   E6POS P1_B_1_App1Place={X 696.23437,Y 929.21517,Z 986.29988,A -180,B 0,C -180,S 2,T 2,E1 0,E2 0,E3 0,E4 0,E5 0,E6 0}
   E6POS P1_B_1_App2Place={X 696.23427,Y 929.21551,Z 786.30015,A -180,B 0,C 180,S 2,T 2,E1 0,E2 0,E3 0,E4 0,E5 0,E6 0}
   E6POS P1_B_1_Place={X 567.29912,Y 1052.67757,Z 666.29996,A -180,B 0,C 180,S 2,T 18,E1 0,E2 0,E3 0,E4 0,E5 0,E6 0}
   E6POS P1_B_2_App1Place={X 562.37046,Y 346.47969,Z 986.29988,A -180,B 0,C 180,S 2,T 2,E1 0,E2 0,E3 0,E4 0,E5 0,E6 0}
   E6POS P1_B_2_App2Place={X 562.37047,Y 346.47964,Z 786.30015,A -180,B 0,C 180,S 2,T 2,E1 0,E2 0,E3 0,E4 0,E5 0,E6 0}
   E6POS P1_B_2_Place={X 433.43516,Y 269.94251,Z 666.29996,A -180,B 0,C -180,S 2,T 2,E1 0,E2 0,E3 0,E4 0,E5 0,E6 0}
   E6POS P1_B_3_App1Place={X 4.05134,Y 173.92954,Z 986.29988,A 90,B 0,C 180,S 2,T 2,E1 0,E2 0,E3 0,E4 0,E5 0,E6 0}
   E6POS P1_B_3_App2Place={X 4.05139,Y 177.15339,Z 786.30015,A 90,B 0,C 180,S 2,T 2,E1 0,E2 0,E3 0,E4 0,E5 0,E6 0}
   E6POS P1_B_3_Place={X 134.71509,Y 273.89023,Z 666.29996,A 90,B 0,C 180,S 2,T 2,E1 0,E2 0,E3 0,E4 0,E5 0,E6 0}
   E6POS P1_B_4_App1Place={X 1006.46519,Y 1126.41051,Z 986.29988,A -90,B 0,C -180,S 2,T 2,E1 0,E2 0,E3 0,E4 0,E5 0,E6 0}
   E6POS P1_B_4_App2Place={X 1006.46535,Y 1126.41022,Z 786.30015,A -90,B 0,C 180,S 2,T 2,E1 0,E2 0,E3 0,E4 0,E5 0,E6 0}
   E6POS P1_B_4_Place={X 866.11759,Y 921.41578,Z 666.29996,A -90,B 0,C -180,S 2,T 2,E1 0,E2 0,E3 0,E4 0,E5 0,E6 0}
   E6POS P1_B_5_App1Place={X 696.22107,Y 346.20666,Z 986.29988,A -180,B 0,C -180,S 2,T 2,E1 0,E2 0,E3 0,E4 0,E5 0,E6 0}
   E6POS P1_B_5_App2Place={X 696.22108,Y 346.20663,Z 786.30015,A -180,B 0,C 180,S 2,T 2,E1 0,E2 0,E3 0,E4 0,E5 0,E6 0}
   E6POS P1_B_5_Place={X 567.29973,Y 269.67394,Z 666.29996,A -180,B 0,C 180,S 2,T 2,E1 0,E2 0,E3 0,E4 0,E5 0,E6 0}
   E6POS P1_B_6_App1Place={X 562.36978,Y 929.48243,Z 986.29988,A -180,B 0,C 180,S 2,T 2,E1 0,E2 0,E3 0,E4 0,E5 0,E6 0}
   E6POS P1_B_6_App2Place={X 562.36973,Y 929.48268,Z 786.30015,A -180,B 0,C -180,S 2,T 2,E1 0,E2 0,E3 0,E4 0,E5 0,E6 0}
   E6POS P1_B_6_Place={X 433.43554,Y 1052.93855,Z 666.29996,A -180,B 0,C 180,S 2,T 2,E1 0,E2 0,E3 0,E4 0,E5 0,E6 0}
   E6POS P1_B_7_App1Place={X 30.66561,Y 1051.60347,Z 986.29988,A -90,B 0,C 180,S 2,T 2,E1 0,E2 0,E3 0,E4 0,E5 0,E6 0}
   E6POS P1_B_7_App2Place={X 30.66561,Y 1051.60341,Z 786.30015,A -90,B 0,C 180,S 2,T 2,E1 0,E2 0,E3 0,E4 0,E5 0,E6 0}
   E6POS P1_B_7_Place={X 175.26087,Y 921.40676,Z 666.29996,A -90,B 0,C 180,S 2,T 2,E1 0,E2 0,E3 0,E4 0,E5 0,E6 0}
   E6POS P1_B_8_App1Place={X 955.95654,Y 159.58068,Z 986.29988,A 90,B 0,C 180,S 2,T 34,E1 0,E2 0,E3 0,E4 0,E5 0,E6 0}
   E6POS P1_B_8_App2Place={X 955.95654,Y 159.58069,Z 786.30015,A 90,B 0,C 180,S 2,T 34,E1 0,E2 0,E3 0,E4 0,E5 0,E6 0}
   E6POS P1_B_8_Place={X 825.57189,Y 273.90166,Z 666.29996,A 90,B 0,C 180,S 2,T 34,E1 0,E2 0,E3 0,E4 0,E5 0,E6 0}

   ;ENDFOLD
   ;FOLD  MosaicoC1_Pallet1

   E6POS P1_C1_1_App1Place={X 585.89482,Y 217.99128,Z 986.28312,A -180,B 0,C -180,S 2,T 2,E1 0,E2 0,E3 0,E4 0,E5 0,E6 0}
   E6POS P1_C1_1_App2Place={X 585.89477,Y 217.99161,Z 836.28257,A -180,B 0,C 180,S 2,T 2,E1 0,E2 0,E3 0,E4 0,E5 0,E6 0}
   E6POS P1_C1_1_Place={X 512.66253,Y 90.04064,Z 666.30129,A -180,B 0,C -180,S 2,T 2,E1 0,E2 0,E3 0,E4 0,E5 0,E6 0}
   E6POS P1_C1_2_App1Place={X 585.89508,Y 456.99119,Z 986.28312,A 180,B 0,C 180,S 2,T 2,E1 0,E2 0,E3 0,E4 0,E5 0,E6 0}
   E6POS P1_C1_2_App2Place={X 585.89505,Y 456.99134,Z 836.28257,A -180,B 0,C -180,S 2,T 2,E1 0,E2 0,E3 0,E4 0,E5 0,E6 0}
   E6POS P1_C1_2_Place={X 512.66375,Y 329.04071,Z 666.30129,A -180,B 0,C 180,S 2,T 2,E1 0,E2 0,E3 0,E4 0,E5 0,E6 0}
   E6POS P1_C1_3_App1Place={X 606.92676,Y 689.18267,Z 986.28312,A -180,B 0,C -180,S 2,T 2,E1 0,E2 0,E3 0,E4 0,E5 0,E6 0}
   E6POS P1_C1_3_App2Place={X 606.92684,Y 689.18232,Z 836.28257,A -180,B 0,C 180,S 2,T 2,E1 0,E2 0,E3 0,E4 0,E5 0,E6 0}
   E6POS P1_C1_3_Place={X 537.74298,Y 568.04115,Z 666.30129,A -180,B 0,C 180,S 2,T 2,E1 0,E2 0,E3 0,E4 0,E5 0,E6 0}
   E6POS P1_C1_4_App1Place={X 606.92634,Y 1021.18263,Z 986.28312,A 180,B 0,C -180,S 2,T 2,E1 0,E2 0,E3 0,E4 0,E5 0,E6 0}
   E6POS P1_C1_4_App2Place={X 606.92631,Y 1021.18275,Z 836.28257,A -180,B 0,C -180,S 2,T 2,E1 0,E2 0,E3 0,E4 0,E5 0,E6 0}
   E6POS P1_C1_4_Place={X 537.74306,Y 900.04115,Z 666.30129,A -180,B 0,C -180,S 2,T 18,E1 0,E2 0,E3 0,E4 0,E5 0,E6 0}
   E6POS P1_C1_5_App1Place={X 606.2009,Y 212.00378,Z 986.28312,A -180,B 0,C -180,S 2,T 2,E1 0,E2 0,E3 0,E4 0,E5 0,E6 0}
   E6POS P1_C1_5_App2Place={X 606.20094,Y 212.00353,Z 836.28257,A -180,B 0,C -180,S 2,T 2,E1 0,E2 0,E3 0,E4 0,E5 0,E6 0}
   E6POS P1_C1_5_Place={X 539.21738,Y 90.04103,Z 666.30129,A -180,B 0,C 180,S 2,T 2,E1 0,E2 0,E3 0,E4 0,E5 0,E6 0}
   E6POS P1_C1_6_App1Place={X 606.20038,Y 544.00374,Z 986.28312,A 180,B 0,C 180,S 2,T 2,E1 0,E2 0,E3 0,E4 0,E5 0,E6 0}
   E6POS P1_C1_6_App2Place={X 606.20036,Y 544.00384,Z 836.28257,A -180,B 0,C 180,S 2,T 2,E1 0,E2 0,E3 0,E4 0,E5 0,E6 0}
   E6POS P1_C1_6_Place={X 539.2172,Y 422.04157,Z 666.30129,A -180,B 0,C 180,S 2,T 2,E1 0,E2 0,E3 0,E4 0,E5 0,E6 0}
   E6POS P1_C1_7_App1Place={X 516.90957,Y 854.03849,Z 986.28312,A 180,B 0,C -180,S 2,T 2,E1 0,E2 0,E3 0,E4 0,E5 0,E6 0}
   E6POS P1_C1_7_App2Place={X 516.9096,Y 854.03829,Z 836.28257,A -180,B 0,C 180,S 2,T 2,E1 0,E2 0,E3 0,E4 0,E5 0,E6 0}
   E6POS P1_C1_7_Place={X 516.90992,Y 754.0383,Z 666.30129,A -180,B 0,C -180,S 2,T 2,E1 0,E2 0,E3 0,E4 0,E5 0,E6 0}
   E6POS P1_C1_8_App1Place={X 516.90957,Y 1093.03906,Z 986.28312,A -180,B 0,C -180,S 2,T 2,E1 0,E2 0,E3 0,E4 0,E5 0,E6 0}
   E6POS P1_C1_8_App2Place={X 516.90967,Y 1093.03859,Z 836.28257,A -180,B 0,C 180,S 2,T 2,E1 0,E2 0,E3 0,E4 0,E5 0,E6 0}
   E6POS P1_C1_8_Place={X 516.90982,Y 993.03884,Z 666.30129,A -180,B 0,C -180,S 2,T 2,E1 0,E2 0,E3 0,E4 0,E5 0,E6 0}

   ;ENDFOLD
   ;FOLD  MosaicoE1_Pallet1

   E6POS P1_E1_1_App1Place={X 194.85126,Y 240.03141,Z 993.17126,A 90,B 0,C 180,S 2,T 2,E1 0,E2 0,E3 0,E4 0,E5 0,E6 0}
   E6POS P1_E1_1_App2Place={X 194.85179,Y 240.03149,Z 843.1711,A 90,B 0,C 180,S 2,T 2,E1 0,E2 0,E3 0,E4 0,E5 0,E6 0}
   E6POS P1_E1_1_Place={X 73.35816,Y 240.03167,Z 690.47496,A 90,B 0,C 180,S 2,T 2,E1 0,E2 0,E3 0,E4 0,E5 0,E6 0}
   E6POS P1_E1_2_App1Place={X 522.85183,Y 240.03135,Z 993.17126,A 90,B 0,C 180,S 2,T 34,E1 0,E2 0,E3 0,E4 0,E5 0,E6 0}
   E6POS P1_E1_2_App2Place={X 522.85174,Y 240.03121,Z 843.1711,A 90,B 0,C 180,S 2,T 34,E1 0,E2 0,E3 0,E4 0,E5 0,E6 0}
   E6POS P1_E1_2_Place={X 401.35813,Y 240.03144,Z 690.47496,A 90,B 0,C 180,S 2,T 34,E1 0,E2 0,E3 0,E4 0,E5 0,E6 0}
   E6POS P1_E1_3_App1Place={X 850.85178,Y 240.03166,Z 993.17126,A 90,B 0,C 180,S 2,T 34,E1 0,E2 0,E3 0,E4 0,E5 0,E6 0}
   E6POS P1_E1_3_App2Place={X 850.85169,Y 240.03128,Z 843.1711,A 90,B 0,C 180,S 2,T 34,E1 0,E2 0,E3 0,E4 0,E5 0,E6 0}
   E6POS P1_E1_3_Place={X 729.35887,Y 240.0316,Z 690.47496,A 90,B 0,C 180,S 2,T 34,E1 0,E2 0,E3 0,E4 0,E5 0,E6 0}
   E6POS P1_E1_4_App1Place={X 622.32094,Y 1010.79553,Z 993.17126,A -180,B 0,C -180,S 2,T 2,E1 0,E2 0,E3 0,E4 0,E5 0,E6 0}
   E6POS P1_E1_4_App2Place={X 622.32108,Y 1010.79584,Z 843.1711,A -180,B 0,C 180,S 2,T 18,E1 0,E2 0,E3 0,E4 0,E5 0,E6 0}
   E6POS P1_E1_4_Place={X 622.32108,Y 907.44031,Z 690.47496,A -180,B 0,C 180,S 2,T 2,E1 0,E2 0,E3 0,E4 0,E5 0,E6 0}
   E6POS P1_E1_5_App1Place={X 622.32111,Y 907.44046,Z 993.17126,A -180,B 0,C 180,S 2,T 2,E1 0,E2 0,E3 0,E4 0,E5 0,E6 0}
   E6POS P1_E1_5_App2Place={X 676.32064,Y 907.52752,Z 843.1711,A -180,B 0,C 180,S 2,T 2,E1 0,E2 0,E3 0,E4 0,E5 0,E6 0}
   E6POS P1_E1_5_Place={X 676.32052,Y 907.52694,Z 690.47496,A -180,B 0,C 180,S 2,T 2,E1 0,E2 0,E3 0,E4 0,E5 0,E6 0}
   E6POS P1_E1_6_App1Place={X 676.32064,Y 907.52752,Z 993.17126,A -180,B 0,C 180,S 2,T 2,E1 0,E2 0,E3 0,E4 0,E5 0,E6 0}
   E6POS P1_E1_6_App2Place={X 730.3205,Y 907.52691,Z 843.1711,A -180,B 0,C 180,S 2,T 2,E1 0,E2 0,E3 0,E4 0,E5 0,E6 0}
   E6POS P1_E1_6_Place={X 730.32055,Y 907.52712,Z 690.47496,A -180,B 0,C 180,S 2,T 2,E1 0,E2 0,E3 0,E4 0,E5 0,E6 0}
   E6POS P1_E1_7_App1Place={X 730.3205,Y 907.52691,Z 993.17126,A -180,B 0,C 180,S 2,T 2,E1 0,E2 0,E3 0,E4 0,E5 0,E6 0}
   E6POS P1_E1_7_App2Place={X 784.32058,Y 907.52713,Z 843.1711,A -180,B 0,C 180,S 2,T 2,E1 0,E2 0,E3 0,E4 0,E5 0,E6 0}
   E6POS P1_E1_7_Place={X 784.32065,Y 907.52737,Z 690.47496,A -180,B 0,C 180,S 2,T 2,E1 0,E2 0,E3 0,E4 0,E5 0,E6 0}
   E6POS P1_E1_8_App1Place={X 624.31165,Y 190.79546,Z 993.17126,A -180,B 0,C 180,S 2,T 2,E1 0,E2 0,E3 0,E4 0,E5 0,E6 0}
   E6POS P1_E1_8_App2Place={X 624.31125,Y 190.79541,Z 843.1711,A -180,B 0,C 180,S 2,T 2,E1 0,E2 0,E3 0,E4 0,E5 0,E6 0}

   E6POS P1_E1_8_Place={X 624.31203,Y 87.43905,Z 690.47496,A -180,B 0,C 180,S 2,T 2,E1 0,E2 0,E3 0,E4 0,E5 0,E6 0}
   E6POS P1_E1_9_App1Place={X 624.31193,Y 87.4387,Z 993.17126,A -180,B 0,C 180,S 2,T 2,E1 0,E2 0,E3 0,E4 0,E5 0,E6 0}
   E6POS P1_E1_9_App2Place={X 678.31177,Y 87.43866,Z 843.1711,A -180,B 0,C 180,S 2,T 2,E1 0,E2 0,E3 0,E4 0,E5 0,E6 0}

   E6POS P1_E1_9_Place={X 678.31185,Y 87.43891,Z 690.47496,A -180,B 0,C -180,S 2,T 2,E1 0,E2 0,E3 0,E4 0,E5 0,E6 0}
   E6POS P1_E1_10_App1Place={X 678.31177,Y 87.43866,Z 993.17126,A -180,B 0,C 180,S 2,T 2,E1 0,E2 0,E3 0,E4 0,E5 0,E6 0}
   E6POS P1_E1_10_App2Place={X 732.31118,Y 87.43893,Z 843.1711,A -180,B 0,C 180,S 2,T 2,E1 0,E2 0,E3 0,E4 0,E5 0,E6 0}

   E6POS P1_E1_10_Place={X 732.31137,Y 87.43945,Z 690.47496,A -180,B 0,C 180,S 2,T 2,E1 0,E2 0,E3 0,E4 0,E5 0,E6 0}
   E6POS P1_E1_11_App1Place={X 732.31118,Y 87.43893,Z 993.17126,A -180,B 0,C 180,S 2,T 2,E1 0,E2 0,E3 0,E4 0,E5 0,E6 0}
   E6POS P1_E1_11_App2Place={X 786.31144,Y 87.43887,Z 843.1711,A -180,B 0,C -180,S 2,T 2,E1 0,E2 0,E3 0,E4 0,E5 0,E6 0}

   E6POS P1_E1_11_Place={X 786.31151,Y 87.43905,Z 690.47496,A -180,B 0,C -180,S 2,T 2,E1 0,E2 0,E3 0,E4 0,E5 0,E6 0}
   E6POS P1_E1_12_App1Place={X 838.55884,Y 1064.39297,Z 993.17126,A -90,B 0,C -180,S 2,T 2,E1 0,E2 0,E3 0,E4 0,E5 0,E6 0}
   E6POS P1_E1_12_App2Place={X 838.55901,Y 1064.39353,Z 843.1711,A -90,B 0,C 180,S 2,T 2,E1 0,E2 0,E3 0,E4 0,E5 0,E6 0}

   E6POS P1_E1_12_Place={X 938.55894,Y 964.39354,Z 690.47496,A -90,B 0,C 180,S 2,T 2,E1 0,E2 0,E3 0,E4 0,E5 0,E6 0}
   E6POS P1_E1_13_App1Place={X 510.55787,Y 1064.39363,Z 993.17126,A -89.99997,B 0,C 180,S 2,T 2,E1 0,E2 0,E3 0,E4 0,E5 0,E6 0}
   E6POS P1_E1_13_App2Place={X 510.55802,Y 1064.39347,Z 843.1711,A -89.99997,B 0,C 180,S 2,T 2,E1 0,E2 0,E3 0,E4 0,E5 0,E6 0}

   E6POS P1_E1_13_Place={X 610.5583,Y 964.39342,Z 690.47496,A -89.99997,B 0,C 180,S 2,T 2,E1 0,E2 0,E3 0,E4 0,E5 0,E6 0}
   E6POS P1_E1_14_App1Place={X 182.55908,Y 1064.39364,Z 993.17126,A -90,B 0,C 180,S 2,T 2,E1 0,E2 0,E3 0,E4 0,E5 0,E6 0}
   E6POS P1_E1_14_App2Place={X 182.55871,Y 1064.39336,Z 843.1711,A -90,B 0,C 180,S 2,T 2,E1 0,E2 0,E3 0,E4 0,E5 0,E6 0}

   E6POS P1_E1_14_Place={X 282.55806,Y 964.39307,Z 690.47496,A -89.99997,B 0,C 180,S 2,T 2,E1 0,E2 0,E3 0,E4 0,E5 0,E6 0}

   ;ENDFOLD
   ;FOLD  MosaicoE2_Pallet1

   E6POS P1_E2_1_App1Place={X 194.85126,Y 240.03141,Z 953.17126,A 90,B 0,C 180,S 2,T 2,E1 0,E2 0,E3 0,E4 0,E5 0,E6 0}
   E6POS P1_E2_1_App2Place={X 194.85179,Y 240.03149,Z 803.1711,A 90,B 0,C 180,S 2,T 2,E1 0,E2 0,E3 0,E4 0,E5 0,E6 0}
   E6POS P1_E2_1_Place={X 73.35816,Y 240.03167,Z 650.47496,A 90,B 0,C 180,S 2,T 2,E1 0,E2 0,E3 0,E4 0,E5 0,E6 0}
   E6POS P1_E2_2_App1Place={X 522.85183,Y 240.03135,Z 953.17126,A 90,B 0,C 180,S 2,T 34,E1 0,E2 0,E3 0,E4 0,E5 0,E6 0}
   E6POS P1_E2_2_App2Place={X 522.85174,Y 240.03121,Z 803.1711,A 90,B 0,C 180,S 2,T 34,E1 0,E2 0,E3 0,E4 0,E5 0,E6 0}
   E6POS P1_E2_2_Place={X 401.35813,Y 240.03144,Z 650.47496,A 90,B 0,C 180,S 2,T 34,E1 0,E2 0,E3 0,E4 0,E5 0,E6 0}
   E6POS P1_E2_3_App1Place={X 850.85178,Y 240.03166,Z 953.17126,A 90,B 0,C 180,S 2,T 34,E1 0,E2 0,E3 0,E4 0,E5 0,E6 0}
   E6POS P1_E2_3_App2Place={X 850.85169,Y 240.03128,Z 803.1711,A 90,B 0,C 180,S 2,T 34,E1 0,E2 0,E3 0,E4 0,E5 0,E6 0}
   E6POS P1_E2_3_Place={X 729.35887,Y 240.0316,Z 650.47496,A 90,B 0,C 180,S 2,T 34,E1 0,E2 0,E3 0,E4 0,E5 0,E6 0}
   E6POS P1_E2_4_App1Place={X 622.32094,Y 1010.79553,Z 953.17126,A -180,B 0,C -180,S 2,T 2,E1 0,E2 0,E3 0,E4 0,E5 0,E6 0}
   E6POS P1_E2_4_App2Place={X 622.32108,Y 1010.79584,Z 803.1711,A -180,B 0,C 180,S 2,T 18,E1 0,E2 0,E3 0,E4 0,E5 0,E6 0}
   E6POS P1_E2_4_Place={X 622.32108,Y 907.44031,Z 650.47496,A -180,B 0,C 180,S 2,T 18,E1 0,E2 0,E3 0,E4 0,E5 0,E6 0}
   E6POS P1_E2_5_App1Place={X 622.32111,Y 907.44046,Z 953.17126,A -180,B 0,C 180,S 2,T 2,E1 0,E2 0,E3 0,E4 0,E5 0,E6 0}
   E6POS P1_E2_5_App2Place={X 676.32064,Y 907.52752,Z 803.1711,A -180,B 0,C 180,S 2,T 2,E1 0,E2 0,E3 0,E4 0,E5 0,E6 0}
   E6POS P1_E2_5_Place={X 676.32052,Y 907.52694,Z 650.47496,A -180,B 0,C 180,S 2,T 18,E1 0,E2 0,E3 0,E4 0,E5 0,E6 0}
   E6POS P1_E2_6_App1Place={X 676.32064,Y 907.52752,Z 953.17126,A -180,B 0,C 180,S 2,T 2,E1 0,E2 0,E3 0,E4 0,E5 0,E6 0}
   E6POS P1_E2_6_App2Place={X 730.3205,Y 907.52691,Z 803.1711,A -180,B 0,C 180,S 2,T 2,E1 0,E2 0,E3 0,E4 0,E5 0,E6 0}
   E6POS P1_E2_6_Place={X 730.32055,Y 907.52712,Z 650.47496,A -180,B 0,C 180,S 2,T 2,E1 0,E2 0,E3 0,E4 0,E5 0,E6 0}
   E6POS P1_E2_7_App1Place={X 730.3205,Y 907.52691,Z 953.17126,A -180,B 0,C 180,S 2,T 2,E1 0,E2 0,E3 0,E4 0,E5 0,E6 0}
   E6POS P1_E2_7_App2Place={X 784.32058,Y 907.52713,Z 803.1711,A -180,B 0,C 180,S 2,T 2,E1 0,E2 0,E3 0,E4 0,E5 0,E6 0}
   E6POS P1_E2_7_Place={X 784.32065,Y 907.52737,Z 650.47496,A -180,B 0,C 180,S 2,T 2,E1 0,E2 0,E3 0,E4 0,E5 0,E6 0}
   E6POS P1_E2_8_App1Place={X 624.31165,Y 190.79546,Z 953.17126,A -180,B 0,C 180,S 2,T 2,E1 0,E2 0,E3 0,E4 0,E5 0,E6 0}
   E6POS P1_E2_8_App2Place={X 624.31125,Y 190.79541,Z 803.1711,A -180,B 0,C 180,S 2,T 2,E1 0,E2 0,E3 0,E4 0,E5 0,E6 0}
   E6POS P1_E2_8_Place={X 624.31203,Y 87.43905,Z 650.47496,A -180,B 0,C 180,S 2,T 2,E1 0,E2 0,E3 0,E4 0,E5 0,E6 0}
   E6POS P1_E2_9_App1Place={X 624.31193,Y 87.4387,Z 953.17126,A -180,B 0,C 180,S 2,T 2,E1 0,E2 0,E3 0,E4 0,E5 0,E6 0}
   E6POS P1_E2_9_App2Place={X 678.31177,Y 87.43866,Z 803.1711,A -180,B 0,C 180,S 2,T 2,E1 0,E2 0,E3 0,E4 0,E5 0,E6 0}
   E6POS P1_E2_9_Place={X 678.31185,Y 87.43891,Z 650.47496,A -180,B 0,C -180,S 2,T 2,E1 0,E2 0,E3 0,E4 0,E5 0,E6 0}
   E6POS P1_E2_10_App1Place={X 678.31177,Y 87.43866,Z 953.17126,A -180,B 0,C 180,S 2,T 2,E1 0,E2 0,E3 0,E4 0,E5 0,E6 0}
   E6POS P1_E2_10_App2Place={X 732.31118,Y 87.43893,Z 803.1711,A -180,B 0,C 180,S 2,T 2,E1 0,E2 0,E3 0,E4 0,E5 0,E6 0}
   E6POS P1_E2_10_Place={X 732.31137,Y 87.43945,Z 650.47496,A -180,B 0,C 180,S 2,T 2,E1 0,E2 0,E3 0,E4 0,E5 0,E6 0}
   E6POS P1_E2_11_App1Place={X 732.31118,Y 87.43893,Z 953.17126,A -180,B 0,C 180,S 2,T 2,E1 0,E2 0,E3 0,E4 0,E5 0,E6 0}
   E6POS P1_E2_11_App2Place={X 786.31144,Y 87.43887,Z 803.1711,A -180,B 0,C -180,S 2,T 2,E1 0,E2 0,E3 0,E4 0,E5 0,E6 0}
   E6POS P1_E2_11_Place={X 786.31151,Y 87.43905,Z 650.47496,A -180,B 0,C -180,S 2,T 2,E1 0,E2 0,E3 0,E4 0,E5 0,E6 0}
   E6POS P1_E2_12_App1Place={X 838.55884,Y 1064.39297,Z 953.17126,A -90,B 0,C -180,S 2,T 2,E1 0,E2 0,E3 0,E4 0,E5 0,E6 0}
   E6POS P1_E2_12_App2Place={X 838.55901,Y 1064.39353,Z 803.1711,A -90,B 0,C 180,S 2,T 2,E1 0,E2 0,E3 0,E4 0,E5 0,E6 0}

   E6POS P1_E2_12_Place={X 938.55894,Y 964.39354,Z 650.47496,A -90,B 0,C 180,S 2,T 2,E1 0,E2 0,E3 0,E4 0,E5 0,E6 0}
   E6POS P1_E2_13_App1Place={X 510.55787,Y 1064.39363,Z 953.17126,A -89.99997,B 0,C 180,S 2,T 2,E1 0,E2 0,E3 0,E4 0,E5 0,E6 0}
   E6POS P1_E2_13_App2Place={X 510.55802,Y 1064.39347,Z 803.1711,A -89.99997,B 0,C 180,S 2,T 2,E1 0,E2 0,E3 0,E4 0,E5 0,E6 0}

   E6POS P1_E2_13_Place={X 610.5583,Y 964.39342,Z 650.47496,A -89.99997,B 0,C 180,S 2,T 2,E1 0,E2 0,E3 0,E4 0,E5 0,E6 0}
   E6POS P1_E2_14_App1Place={X 182.55908,Y 1064.39364,Z 953.17126,A -90,B 0,C 180,S 2,T 2,E1 0,E2 0,E3 0,E4 0,E5 0,E6 0}
   E6POS P1_E2_14_App2Place={X 182.55871,Y 1064.39336,Z 803.1711,A -90,B 0,C 180,S 2,T 2,E1 0,E2 0,E3 0,E4 0,E5 0,E6 0}

   E6POS P1_E2_14_Place={X 282.55806,Y 964.39307,Z 650.47496,A -89.99997,B 0,C 180,S 2,T 2,E1 0,E2 0,E3 0,E4 0,E5 0,E6 0}

   ;ENDFOLD
   ;FOLD  MosaicoF_Pallet1

   E6POS P1_F_1_App1Place={X 185.70996,Y 503.84704,Z 990.17104,A -89.99997,B 0,C 180,S 2,T 2,E1 0,E2 0,E3 0,E4 0,E5 0,E6 0}
   E6POS P1_F_1_App2Place={X 185.71037,Y 503.84729,Z 840.17131,A -89.99997,B 0,C 180,S 2,T 2,E1 0,E2 0,E3 0,E4 0,E5 0,E6 0}
   E6POS P1_F_1_Place={X 59.05642,Y 604.23198,Z 654.93708,A -89.99997,B 0,C 180,S 2,T 2,E1 0,E2 0,E3 0,E4 0,E5 0,E6 0}
   E6POS P1_F_2_App1Place={X 484.71014,Y 503.84728,Z 990.17104,A -89.99997,B 0,C 180,S 2,T 2,E1 0,E2 0,E3 0,E4 0,E5 0,E6 0}
   E6POS P1_F_2_App2Place={X 484.71027,Y 503.84725,Z 840.17131,A -89.99997,B 0,C 180,S 2,T 2,E1 0,E2 0,E3 0,E4 0,E5 0,E6 0}
   E6POS P1_F_2_Place={X 358.05527,Y 604.23504,Z 654.93708,A -89.99997,B 0,C 180,S 2,T 2,E1 0,E2 0,E3 0,E4 0,E5 0,E6 0}
   E6POS P1_F_3_App1Place={X 783.33985,Y 500.30966,Z 990.17104,A -90,B 0,C 180,S 2,T 2,E1 0,E2 0,E3 0,E4 0,E5 0,E6 0}
   E6POS P1_F_3_App2Place={X 783.33995,Y 500.31005,Z 840.17131,A -90,B 0,C 180,S 2,T 2,E1 0,E2 0,E3 0,E4 0,E5 0,E6 0}
   E6POS P1_F_3_Place={X 657.05567,Y 600.73453,Z 654.93708,A -90,B 0,C 180,S 2,T 2,E1 0,E2 0,E3 0,E4 0,E5 0,E6 0}
   E6POS P1_F_4_App1Place={X 981.33967,Y 500.30989,Z 990.17104,A -90,B 0,C 180,S 2,T 2,E1 0,E2 0,E3 0,E4 0,E5 0,E6 0}
   E6POS P1_F_4_App2Place={X 981.33982,Y 500.30975,Z 840.17131,A -90,B 0,C 180,S 2,T 2,E1 0,E2 0,E3 0,E4 0,E5 0,E6 0}
   E6POS P1_F_4_Place={X 855.0547,Y 600.73492,Z 654.93708,A -90,B 0,C 180,S 2,T 2,E1 0,E2 0,E3 0,E4 0,E5 0,E6 0}
   E6POS P1_F_5_App1Place={X 185.3398,Y 495.81009,Z 990.17104,A -90,B 0,C 180,S 2,T 2,E1 0,E2 0,E3 0,E4 0,E5 0,E6 0}
   E6POS P1_F_5_App2Place={X 185.33937,Y 495.81034,Z 840.17131,A -90,B 0,C 180,S 2,T 2,E1 0,E2 0,E3 0,E4 0,E5 0,E6 0}
   E6POS P1_F_5_Place={X 59.05866,Y 596.22286,Z 654.93708,A -90,B 0,C 180,S 2,T 2,E1 0,E2 0,E3 0,E4 0,E5 0,E6 0}
   E6POS P1_F_6_App1Place={X 383.34027,Y 495.81061,Z 990.17104,A -90,B 0,C 180,S 2,T 2,E1 0,E2 0,E3 0,E4 0,E5 0,E6 0}
   E6POS P1_F_6_App2Place={X 383.33973,Y 495.81031,Z 840.17131,A -90,B 0,C 180,S 2,T 2,E1 0,E2 0,E3 0,E4 0,E5 0,E6 0}
   E6POS P1_F_6_Place={X 257.05855,Y 596.22277,Z 654.93708,A -90,B 0,C 180,S 2,T 2,E1 0,E2 0,E3 0,E4 0,E5 0,E6 0}
   E6POS P1_F_7_App1Place={X 581.71086,Y 500.34692,Z 990.17104,A -90,B 0,C 180,S 2,T 2,E1 0,E2 0,E3 0,E4 0,E5 0,E6 0}
   E6POS P1_F_7_App2Place={X 581.71089,Y 500.3468,Z 840.17131,A -90,B 0,C 180,S 2,T 2,E1 0,E2 0,E3 0,E4 0,E5 0,E6 0}
   E6POS P1_F_7_Place={X 455.05485,Y 600.73514,Z 654.93708,A -90,B 0,C 180,S 2,T 2,E1 0,E2 0,E3 0,E4 0,E5 0,E6 0}
   E6POS P1_F_8_App1Place={X 880.71075,Y 500.34652,Z 990.17104,A -90,B 0,C 180,S 2,T 2,E1 0,E2 0,E3 0,E4 0,E5 0,E6 0}
   E6POS P1_F_8_App2Place={X 880.7105,Y 500.34636,Z 840.17131,A -90,B 0,C 180,S 2,T 2,E1 0,E2 0,E3 0,E4 0,E5 0,E6 0}
   E6POS P1_F_8_Place={X 754.05499,Y 600.73496,Z 654.93708,A -90,B 0,C 180,S 2,T 2,E1 0,E2 0,E3 0,E4 0,E5 0,E6 0}

   ;ENDFOLD
   ;FOLD  MosaicoG_Pallet1

   E6POS P1_G_1_App1Place={X 149.3733,Y -2.098,Z 1001.61791,A -90,B 0,C 180,S 2,T 2,E1 0,E2 0,E3 0,E4 0,E5 0,E6 0}
   E6POS P1_G_1_App2Place={X 149.37352,Y -2.09821,Z 851.61778,A -90,B 0,C 180,S 2,T 2,E1 0,E2 0,E3 0,E4 0,E5 0,E6 0}
   E6POS P1_G_1_Place={X 49.37367,Y -2.09846,Z 651.61785,A -90,B 0,C 180,S 2,T 2,E1 0,E2 0,E3 0,E4 0,E5 0,E6 0}
   E6POS P1_G_2_App1Place={X 353.37484,Y 585.90186,Z 1001.61791,A -90,B 0,C 180,S 2,T 2,E1 0,E2 0,E3 0,E4 0,E5 0,E6 0}
   E6POS P1_G_2_App2Place={X 353.37434,Y 585.90171,Z 851.61778,A -90,B 0,C 180,S 2,T 2,E1 0,E2 0,E3 0,E4 0,E5 0,E6 0}
   E6POS P1_G_2_Place={X 253.37397,Y 585.90191,Z 651.61785,A -90,B 0,C 180,S 2,T 2,E1 0,E2 0,E3 0,E4 0,E5 0,E6 0}
   E6POS P1_G_3_App1Place={X 162.41244,Y 1258.69084,Z 1001.61791,A -90,B 0,C 180,S 2,T 18,E1 0,E2 0,E3 0,E4 0,E5 0,E6 0}
   E6POS P1_G_3_App2Place={X 162.41236,Y 1258.69069,Z 851.61778,A -90,B 0,C 180,S 2,T 18,E1 0,E2 0,E3 0,E4 0,E5 0,E6 0}
   E6POS P1_G_3_Place={X 49.37239,Y 1173.90187,Z 651.61785,A -90,B 0,C 180,S 2,T 18,E1 0,E2 0,E3 0,E4 0,E5 0,E6 0}
   E6POS P1_G_4_App1Place={X 559.12256,Y -2.23501,Z 1001.61791,A -90,B 0,C 180,S 2,T 2,E1 0,E2 0,E3 0,E4 0,E5 0,E6 0}
   E6POS P1_G_4_App2Place={X 559.12222,Y -2.235,Z 851.61778,A -90,B 0,C 180,S 2,T 2,E1 0,E2 0,E3 0,E4 0,E5 0,E6 0}
   E6POS P1_G_4_Place={X 457.3734,Y -26.09812,Z 651.61785,A -90,B 0,C 180,S 2,T 2,E1 0,E2 0,E3 0,E4 0,E5 0,E6 0}
   E6POS P1_G_5_App1Place={X 566.40187,Y 1306.30302,Z 1001.61791,A -90,B 0,C 180,S 2,T 18,E1 0,E2 0,E3 0,E4 0,E5 0,E6 0}
   E6POS P1_G_5_App2Place={X 566.4018,Y 1306.30279,Z 851.61778,A -90,B 0,C 180,S 2,T 18,E1 0,E2 0,E3 0,E4 0,E5 0,E6 0}
   E6POS P1_G_5_Place={X 343.37167,Y 1197.90666,Z 651.61785,A -90,B 0,C 180,S 2,T 18,E1 0,E2 0,E3 0,E4 0,E5 0,E6 0}
   E6POS P1_G_6_App1Place={X 770.40189,Y 1306.30308,Z 1001.61791,A -90,B 0,C 180,S 2,T 18,E1 0,E2 0,E3 0,E4 0,E5 0,E6 0}
   E6POS P1_G_6_App2Place={X 770.4018,Y 1306.30279,Z 851.61778,A -90,B 0,C 180,S 2,T 18,E1 0,E2 0,E3 0,E4 0,E5 0,E6 0}
   E6POS P1_G_6_Place={X 547.37167,Y 1197.90666,Z 651.61785,A -90,B 0,C 180,S 2,T 18,E1 0,E2 0,E3 0,E4 0,E5 0,E6 0}
   E6POS P1_G_7_App1Place={X 853.12069,Y 609.77263,Z 1001.61791,A -89.99997,B 0,C 180,S 2,T 2,E1 0,E2 0,E3 0,E4 0,E5 0,E6 0}
   E6POS P1_G_7_App2Place={X 853.12035,Y 609.77308,Z 851.61778,A -89.99997,B 0,C 180,S 2,T 2,E1 0,E2 0,E3 0,E4 0,E5 0,E6 0}
   E6POS P1_G_7_Place={X 751.37887,Y 612.61574,Z 651.61785,A -89.99997,B 0,C 180,S 2,T 2,E1 0,E2 0,E3 0,E4 0,E5 0,E6 0}
   E6POS P1_G_8_App1Place={X 753.12073,Y 609.77254,Z 1001.61791,A -90,B 0,C 180,S 2,T 2,E1 0,E2 0,E3 0,E4 0,E5 0,E6 0}
   E6POS P1_G_8_App2Place={X 753.12006,Y 654.77255,Z 851.61778,A -89.99997,B 0,C 180,S 2,T 2,E1 0,E2 0,E3 0,E4 0,E5 0,E6 0}
   E6POS P1_G_8_Place={X 753.12003,Y 654.77244,Z 651.61785,A -89.99997,B 0,C 180,S 2,T 2,E1 0,E2 0,E3 0,E4 0,E5 0,E6 0}
   E6POS P1_G_9_App1Place={X 753.12006,Y 654.77255,Z 1001.61791,A -89.99997,B 0,C 180,S 2,T 2,E1 0,E2 0,E3 0,E4 0,E5 0,E6 0}
   E6POS P1_G_9_App2Place={X 753.12053,Y 699.77216,Z 851.61778,A -90,B 0,C 180,S 2,T 2,E1 0,E2 0,E3 0,E4 0,E5 0,E6 0}
   E6POS P1_G_9_Place={X 753.12063,Y 699.77251,Z 651.61785,A -90,B 0,C 180,S 2,T 2,E1 0,E2 0,E3 0,E4 0,E5 0,E6 0}
   E6POS P1_G_10_App1Place={X 753.12053,Y 699.77216,Z 1001.61791,A -90,B 0,C 180,S 2,T 2,E1 0,E2 0,E3 0,E4 0,E5 0,E6 0}
   E6POS P1_G_10_App2Place={X 753.12058,Y 744.7725,Z 851.61778,A -90,B 0,C 180,S 2,T 2,E1 0,E2 0,E3 0,E4 0,E5 0,E6 0}
   E6POS P1_G_10_Place={X 753.12059,Y 744.77255,Z 651.61785,A -90,B 0,C 180,S 2,T 2,E1 0,E2 0,E3 0,E4 0,E5 0,E6 0}
   E6POS P1_G_11_App1Place={X 753.12058,Y 744.7725,Z 1001.61791,A -90,B 0,C 180,S 2,T 2,E1 0,E2 0,E3 0,E4 0,E5 0,E6 0}
   E6POS P1_G_11_App2Place={X 753.12054,Y 789.7722,Z 851.61778,A -90,B 0,C 180,S 2,T 2,E1 0,E2 0,E3 0,E4 0,E5 0,E6 0}
   E6POS P1_G_11_Place={X 753.12064,Y 789.7726,Z 651.61785,A -90,B 0,C 180,S 2,T 2,E1 0,E2 0,E3 0,E4 0,E5 0,E6 0}
   E6POS P1_G_12_App1Place={X 443.37216,Y 585.90697,Z 1001.61791,A -90,B 0,C 180,S 2,T 2,E1 0,E2 0,E3 0,E4 0,E5 0,E6 0}
   E6POS P1_G_12_App2Place={X 443.37195,Y 585.90667,Z 851.61778,A -90,B 0,C 180,S 2,T 2,E1 0,E2 0,E3 0,E4 0,E5 0,E6 0}
   E6POS P1_G_12_Place={X 343.37181,Y 585.90688,Z 651.61785,A -90,B 0,C 180,S 2,T 2,E1 0,E2 0,E3 0,E4 0,E5 0,E6 0}
   E6POS P1_G_13_App1Place={X 647.37126,Y -2.09336,Z 1001.61791,A -90,B 0,C 180,S 2,T 2,E1 0,E2 0,E3 0,E4 0,E5 0,E6 0}
   E6POS P1_G_13_App2Place={X 647.37173,Y -2.09348,Z 851.61778,A -90,B 0,C 180,S 2,T 2,E1 0,E2 0,E3 0,E4 0,E5 0,E6 0}
   E6POS P1_G_13_Place={X 547.37181,Y -2.0932,Z 651.61785,A -90,B 0,C 180,S 2,T 2,E1 0,E2 0,E3 0,E4 0,E5 0,E6 0}
   E6POS P1_G_14_App1Place={X 393.37097,Y 1223.9067,Z 1001.61791,A -90,B 0,C 180,S 2,T 2,E1 0,E2 0,E3 0,E4 0,E5 0,E6 0}
   E6POS P1_G_14_App2Place={X 393.37089,Y 1223.90695,Z 851.61778,A -90,B 0,C 180,S 2,T 2,E1 0,E2 0,E3 0,E4 0,E5 0,E6 0}
   E6POS P1_G_14_Place={X 343.37089,Y 1173.90695,Z 651.61785,A -90,B 0,C 180,S 2,T 18,E1 0,E2 0,E3 0,E4 0,E5 0,E6 0}
   E6POS P1_G_15_App1Place={X 853.11893,Y -26.09388,Z 1001.61791,A -90,B 0,C 180,S 2,T 2,E1 0,E2 0,E3 0,E4 0,E5 0,E6 0}
   E6POS P1_G_15_App2Place={X 853.11941,Y -26.09348,Z 851.61778,A -90,B 0,C 180,S 2,T 2,E1 0,E2 0,E3 0,E4 0,E5 0,E6 0}
   E6POS P1_G_15_Place={X 751.37143,Y -26.09385,Z 651.61785,A -90,B 0,C 180,S 2,T 2,E1 0,E2 0,E3 0,E4 0,E5 0,E6 0}
   E6POS P1_G_16_App1Place={X 737.36384,Y 1297.90658,Z 1001.61791,A -90,B 0,C -180,S 2,T 2,E1 0,E2 0,E3 0,E4 0,E5 0,E6 0}
   E6POS P1_G_16_App2Place={X 737.36384,Y 1297.90637,Z 851.61778,A -90,B 0,C 180,S 2,T 2,E1 0,E2 0,E3 0,E4 0,E5 0,E6 0}
   E6POS P1_G_16_Place={X 637.37555,Y 1197.90665,Z 651.61785,A -90,B 0,C 180,S 2,T 18,E1 0,E2 0,E3 0,E4 0,E5 0,E6 0}
   E6POS P1_G_17_App1Place={X 941.36401,Y 1297.9064,Z 1001.61791,A -90,B 0,C 180,S 2,T 2,E1 0,E2 0,E3 0,E4 0,E5 0,E6 0}
   E6POS P1_G_17_App2Place={X 941.36384,Y 1297.90637,Z 851.61778,A -90,B 0,C -180,S 2,T 2,E1 0,E2 0,E3 0,E4 0,E5 0,E6 0}
   E6POS P1_G_17_Place={X 841.37555,Y 1197.90665,Z 651.61785,A -90,B 0,C -180,S 2,T 18,E1 0,E2 0,E3 0,E4 0,E5 0,E6 0}
   E6POS P1_G_18_App1Place={X 75.37301,Y 583.87485,Z 1001.61791,A 90,B 0,C 180,S 2,T 2,E1 0,E2 0,E3 0,E4 0,E5 0,E6 0}
   E6POS P1_G_18_App2Place={X 75.37307,Y 583.87481,Z 851.61778,A 90,B 0,C 180,S 2,T 2,E1 0,E2 0,E3 0,E4 0,E5 0,E6 0}
   E6POS P1_G_18_Place={X 220.62117,Y 583.87476,Z 651.61785,A 90,B 0,C 180,S 2,T 34,E1 0,E2 0,E3 0,E4 0,E5 0,E6 0}
   E6POS P1_G_19_App1Place={X 220.62116,Y 583.87476,Z 1001.61791,A 90,B 0,C 180,S 2,T 34,E1 0,E2 0,E3 0,E4 0,E5 0,E6 0}
   E6POS P1_G_19_App2Place={X 220.62116,Y 538.87476,Z 851.61778,A 90,B 0,C 180,S 2,T 34,E1 0,E2 0,E3 0,E4 0,E5 0,E6 0}
   E6POS P1_G_19_Place={X 220.62116,Y 538.87476,Z 651.61785,A 90,B 0,C 180,S 2,T 34,E1 0,E2 0,E3 0,E4 0,E5 0,E6 0}
   E6POS P1_G_20_App1Place={X 220.62116,Y 538.87476,Z 1001.61791,A 90,B 0,C 180,S 2,T 34,E1 0,E2 0,E3 0,E4 0,E5 0,E6 0}
   E6POS P1_G_20_App2Place={X 220.62116,Y 493.87476,Z 851.61778,A 90,B 0,C 180,S 2,T 34,E1 0,E2 0,E3 0,E4 0,E5 0,E6 0}
   E6POS P1_G_20_Place={X 220.62116,Y 493.87476,Z 651.61785,A 90,B 0,C 180,S 2,T 34,E1 0,E2 0,E3 0,E4 0,E5 0,E6 0}
   E6POS P1_G_21_App1Place={X 220.62116,Y 493.87476,Z 1001.61791,A 90,B 0,C 180,S 2,T 34,E1 0,E2 0,E3 0,E4 0,E5 0,E6 0}
   E6POS P1_G_21_App2Place={X 220.62116,Y 448.87476,Z 851.61778,A 90,B 0,C 180,S 2,T 34,E1 0,E2 0,E3 0,E4 0,E5 0,E6 0}
   E6POS P1_G_21_Place={X 220.62116,Y 448.87476,Z 651.61785,A 90,B 0,C 180,S 2,T 34,E1 0,E2 0,E3 0,E4 0,E5 0,E6 0}
   E6POS P1_G_22_App1Place={X 220.62116,Y 448.87476,Z 1001.61791,A 90,B 0,C 180,S 2,T 34,E1 0,E2 0,E3 0,E4 0,E5 0,E6 0}
   E6POS P1_G_22_App2Place={X 220.62116,Y 403.87476,Z 851.61778,A 90,B 0,C 180,S 2,T 34,E1 0,E2 0,E3 0,E4 0,E5 0,E6 0}
   E6POS P1_G_22_Place={X 220.62116,Y 403.87476,Z 651.61785,A 90,B 0,C 180,S 2,T 34,E1 0,E2 0,E3 0,E4 0,E5 0,E6 0}

   ;ENDFOLD
   ;FOLD  MosaicoI_Pallet1

   E6POS P1_I_1_App1Place={X 246.53091,Y 662.70226,Z 986.30203,A -90,B 0,C 180,S 2,T 2,E1 0,E2 0,E3 0,E4 0,E5 0,E6 0}
   E6POS P1_I_1_App2Place={X 246.53091,Y 662.7025,Z 836.30179,A -90,B 0,C 180,S 2,T 2,E1 0,E2 0,E3 0,E4 0,E5 0,E6 0}
   E6POS P1_I_1_Place={X 120.2419,Y 563.31321,Z 652.09239,A -90,B 0,C 180,S 2,T 2,E1 0,E2 0,E3 0,E4 0,E5 0,E6 0}
   E6POS P1_I_2_App1Place={X 120.24188,Y 563.31279,Z 986.30203,A -90,B 0,C 180,S 2,T 2,E1 0,E2 0,E3 0,E4 0,E5 0,E6 0}
   E6POS P1_I_2_App2Place={X 120.24229,Y 624.31271,Z 836.30179,A -90,B 0,C 180,S 2,T 2,E1 0,E2 0,E3 0,E4 0,E5 0,E6 0}
   E6POS P1_I_2_Place={X 120.24227,Y 624.3123,Z 652.09239,A -90,B 0,C 180,S 2,T 2,E1 0,E2 0,E3 0,E4 0,E5 0,E6 0}
   E6POS P1_I_3_App1Place={X 120.24229,Y 624.31271,Z 986.30203,A -90,B 0,C 180,S 2,T 2,E1 0,E2 0,E3 0,E4 0,E5 0,E6 0}
   E6POS P1_I_3_App2Place={X 120.24194,Y 685.31244,Z 836.30179,A -90,B 0,C 180,S 2,T 2,E1 0,E2 0,E3 0,E4 0,E5 0,E6 0}
   E6POS P1_I_3_Place={X 120.24196,Y 685.31272,Z 652.09239,A -90,B 0,C 180,S 2,T 2,E1 0,E2 0,E3 0,E4 0,E5 0,E6 0}
   E6POS P1_I_4_App1Place={X 584.73524,Y 593.5001,Z 986.30203,A 90,B 0,C -180,S 2,T 34,E1 0,E2 0,E3 0,E4 0,E5 0,E6 0}
   E6POS P1_I_4_App2Place={X 584.73528,Y 593.49987,Z 836.30179,A 90,B 0,C 180,S 2,T 34,E1 0,E2 0,E3 0,E4 0,E5 0,E6 0}
   E6POS P1_I_4_Place={X 484.73518,Y 593.50008,Z 652.09239,A 90,B 0,C 180,S 2,T 34,E1 0,E2 0,E3 0,E4 0,E5 0,E6 0}
   E6POS P1_I_5_App1Place={X 942.73565,Y 593.50042,Z 986.30203,A 90,B 0,C -180,S 2,T 34,E1 0,E2 0,E3 0,E4 0,E5 0,E6 0}
   E6POS P1_I_5_App2Place={X 942.73575,Y 593.50015,Z 836.30179,A 90,B 0,C 180,S 2,T 34,E1 0,E2 0,E3 0,E4 0,E5 0,E6 0}
   E6POS P1_I_5_Place={X 842.73579,Y 593.50005,Z 652.09239,A 90,B 0,C 180,S 2,T 34,E1 0,E2 0,E3 0,E4 0,E5 0,E6 0}
   E6POS P1_I_6_App1Place={X 413.73466,Y 594.42062,Z 986.30203,A 90,B 0,C 180,S 2,T 34,E1 0,E2 0,E3 0,E4 0,E5 0,E6 0}
   E6POS P1_I_6_App2Place={X 413.73463,Y 594.42083,Z 836.30179,A 90,B 0,C 180,S 2,T 34,E1 0,E2 0,E3 0,E4 0,E5 0,E6 0}
   E6POS P1_I_6_Place={X 313.73464,Y 594.42082,Z 652.09239,A 90,B 0,C 180,S 2,T 34,E1 0,E2 0,E3 0,E4 0,E5 0,E6 0}
   E6POS P1_I_7_App1Place={X 771.73426,Y 594.42052,Z 986.30203,A 90,B 0,C -180,S 2,T 34,E1 0,E2 0,E3 0,E4 0,E5 0,E6 0}
   E6POS P1_I_7_App2Place={X 771.73418,Y 594.4208,Z 836.30179,A 90,B 0,C 180,S 2,T 34,E1 0,E2 0,E3 0,E4 0,E5 0,E6 0}
   E6POS P1_I_7_Place={X 671.73443,Y 594.42068,Z 652.09239,A 90,B 0,C 180,S 2,T 34,E1 0,E2 0,E3 0,E4 0,E5 0,E6 0}
   E6POS P1_I_8_App1Place={X 936.24164,Y 563.31281,Z 986.30203,A -90,B 0,C -180,S 2,T 2,E1 0,E2 0,E3 0,E4 0,E5 0,E6 0}
   E6POS P1_I_8_App2Place={X 936.24164,Y 563.31281,Z 836.30179,A -90,B 0,C 180,S 2,T 2,E1 0,E2 0,E3 0,E4 0,E5 0,E6 0}
   E6POS P1_I_8_Place={X 836.24218,Y 563.31266,Z 652.09239,A -90,B 0,C 180,S 2,T 2,E1 0,E2 0,E3 0,E4 0,E5 0,E6 0}
   E6POS P1_I_9_App1Place={X 836.24219,Y 563.31262,Z 986.30203,A -90,B 0,C 180,S 2,T 2,E1 0,E2 0,E3 0,E4 0,E5 0,E6 0}
   E6POS P1_I_9_App2Place={X 836.24173,Y 624.31272,Z 836.30179,A -90,B 0,C 180,S 2,T 2,E1 0,E2 0,E3 0,E4 0,E5 0,E6 0}
   E6POS P1_I_9_Place={X 836.24181,Y 624.31245,Z 652.09239,A -90,B 0,C 180,S 2,T 2,E1 0,E2 0,E3 0,E4 0,E5 0,E6 0}
   E6POS P1_I_10_App1Place={X 836.24173,Y 624.31272,Z 986.30203,A -90,B 0,C 180,S 2,T 2,E1 0,E2 0,E3 0,E4 0,E5 0,E6 0}
   E6POS P1_I_10_App2Place={X 836.24228,Y 685.31292,Z 836.30179,A -90,B 0,C 180,S 2,T 2,E1 0,E2 0,E3 0,E4 0,E5 0,E6 0}
   E6POS P1_I_10_Place={X 836.24232,Y 685.3128,Z 652.09239,A -90,B 0,C 180,S 2,T 2,E1 0,E2 0,E3 0,E4 0,E5 0,E6 0}

   ;ENDFOLD
   ;FOLD  MosaicoJ_Pallet1

   E6POS P1_J_1_App1Place={X 205.12222,Y 673.0107,Z 986.30227,A 90,B 0,C 180,S 2,T 34,E1 0,E2 0,E3 0,E4 0,E5 0,E6 0}
   E6POS P1_J_1_App2Place={X 205.12222,Y 673.01047,Z 786.30223,A 90,B 0,C 180,S 2,T 34,E1 0,E2 0,E3 0,E4 0,E5 0,E6 0}
   E6POS P1_J_1_Place={X 83.2071,Y 563.55362,Z 666.3006,A 90,B 0,C 180,S 2,T 2,E1 0,E2 0,E3 0,E4 0,E5 0,E6 0}
   E6POS P1_J_2_App1Place={X 996.70798,Y 190.44819,Z 986.30227,A -180,B 0,C -180,S 2,T 2,E1 0,E2 0,E3 0,E4 0,E5 0,E6 0}
   E6POS P1_J_2_App2Place={X 996.70793,Y 190.44835,Z 786.30223,A -180,B 0,C 180,S 2,T 2,E1 0,E2 0,E3 0,E4 0,E5 0,E6 0}
   E6POS P1_J_2_Place={X 896.70882,Y 90.44837,Z 666.3006,A -180,B 0,C 180,S 2,T 2,E1 0,E2 0,E3 0,E4 0,E5 0,E6 0}
   E6POS P1_J_3_App1Place={X 996.70887,Y 479.44933,Z 986.30227,A 180,B 0,C -180,S 2,T 2,E1 0,E2 0,E3 0,E4 0,E5 0,E6 0}
   E6POS P1_J_3_App2Place={X 996.70888,Y 479.44931,Z 786.30223,A -180,B 0,C 180,S 2,T 2,E1 0,E2 0,E3 0,E4 0,E5 0,E6 0}
   E6POS P1_J_3_Place={X 896.7079,Y 379.44856,Z 666.3006,A -180,B 0,C -180,S 2,T 2,E1 0,E2 0,E3 0,E4 0,E5 0,E6 0}
   E6POS P1_J_4_App1Place={X 996.70886,Y 768.44899,Z 986.30227,A -180,B 0,C -180,S 2,T 2,E1 0,E2 0,E3 0,E4 0,E5 0,E6 0}
   E6POS P1_J_4_App2Place={X 996.70882,Y 768.44907,Z 786.30223,A -180,B 0,C -180,S 2,T 2,E1 0,E2 0,E3 0,E4 0,E5 0,E6 0}
   E6POS P1_J_4_Place={X 896.708,Y 668.44849,Z 666.3006,A -180,B 0,C -180,S 2,T 2,E1 0,E2 0,E3 0,E4 0,E5 0,E6 0}
   E6POS P1_J_5_App1Place={X 996.70887,Y 1057.44903,Z 986.30227,A 180,B 0,C -180,S 2,T 2,E1 0,E2 0,E3 0,E4 0,E5 0,E6 0}
   E6POS P1_J_5_App2Place={X 996.70891,Y 1057.44895,Z 786.30223,A -180,B 0,C 180,S 2,T 2,E1 0,E2 0,E3 0,E4 0,E5 0,E6 0}
   E6POS P1_J_5_Place={X 896.7083,Y 957.44855,Z 666.3006,A -180,B 0,C 180,S 2,T 2,E1 0,E2 0,E3 0,E4 0,E5 0,E6 0}
   E6POS P1_J_6_App1Place={X 624.70886,Y 190.44877,Z 986.30227,A -180,B 0,C -180,S 2,T 2,E1 0,E2 0,E3 0,E4 0,E5 0,E6 0}
   E6POS P1_J_6_App2Place={X 624.70884,Y 190.44885,Z 786.30223,A -180,B 0,C 180,S 2,T 2,E1 0,E2 0,E3 0,E4 0,E5 0,E6 0}
   E6POS P1_J_6_Place={X 624.70888,Y 90.44835,Z 666.3006,A -180,B 0,C 180,S 2,T 2,E1 0,E2 0,E3 0,E4 0,E5 0,E6 0}
   E6POS P1_J_7_App1Place={X 624.70798,Y 479.44853,Z 986.30227,A -180,B 0,C -180,S 2,T 2,E1 0,E2 0,E3 0,E4 0,E5 0,E6 0}
   E6POS P1_J_7_App2Place={X 624.70799,Y 479.4485,Z 786.30223,A -180,B 0,C -180,S 2,T 2,E1 0,E2 0,E3 0,E4 0,E5 0,E6 0}
   E6POS P1_J_7_Place={X 624.70786,Y 379.44821,Z 666.3006,A -180,B 0,C 180,S 2,T 2,E1 0,E2 0,E3 0,E4 0,E5 0,E6 0}
   E6POS P1_J_8_App1Place={X 624.70824,Y 768.4485,Z 986.30227,A 180,B 0,C 180,S 2,T 2,E1 0,E2 0,E3 0,E4 0,E5 0,E6 0}
   E6POS P1_J_8_App2Place={X 624.70825,Y 768.44844,Z 786.30223,A -180,B 0,C 180,S 2,T 2,E1 0,E2 0,E3 0,E4 0,E5 0,E6 0}
   E6POS P1_J_8_Place={X 624.70846,Y 668.44829,Z 666.3006,A -180,B 0,C -180,S 2,T 2,E1 0,E2 0,E3 0,E4 0,E5 0,E6 0}
   E6POS P1_J_9_App1Place={X 624.70848,Y 1057.44882,Z 986.30227,A 180,B 0,C 180,S 2,T 2,E1 0,E2 0,E3 0,E4 0,E5 0,E6 0}
   E6POS P1_J_9_App2Place={X 624.70849,Y 1057.44878,Z 786.30223,A -180,B 0,C 180,S 2,T 2,E1 0,E2 0,E3 0,E4 0,E5 0,E6 0}
   E6POS P1_J_9_Place={X 624.7086,Y 957.44847,Z 666.3006,A -180,B 0,C 180,S 2,T 2,E1 0,E2 0,E3 0,E4 0,E5 0,E6 0}
   E6POS P1_J_10_App1Place={X 867.21032,Y 562.58543,Z 986.30227,A 90,B 0,C 180,S 2,T 34,E1 0,E2 0,E3 0,E4 0,E5 0,E6 0}
   E6POS P1_J_10_App2Place={X 867.21029,Y 562.58552,Z 786.30223,A 90,B 0,C 180,S 2,T 34,E1 0,E2 0,E3 0,E4 0,E5 0,E6 0}
   E6POS P1_J_10_Place={X 767.21058,Y 562.5858,Z 666.3006,A 90,B 0,C 180,S 2,T 34,E1 0,E2 0,E3 0,E4 0,E5 0,E6 0}

   ;ENDFOLD
   ;FOLD  MosaicoK_Pallet1

   E6POS P1_K_1_App1Place={X 965.18934,Y 160.47355,Z 1002.77226,A -180,B 0,C -180,S 2,T 2,E1 0,E2 0,E3 0,E4 0,E5 0,E6 0}
   E6POS P1_K_1_App2Place={X 965.18946,Y 160.47317,Z 802.77226,A -180,B 0,C 180,S 2,T 2,E1 0,E2 0,E3 0,E4 0,E5 0,E6 0}
   E6POS P1_K_1_Place={X 965.18981,Y 60.47307,Z 652.77183,A -180,B 0,C -180,S 2,T 2,E1 0,E2 0,E3 0,E4 0,E5 0,E6 0}
   E6POS P1_K_2_App1Place={X 289.34828,Y 416.70469,Z 1002.77226,A -180,B 0,C -180,S 2,T 2,E1 0,E2 0,E3 0,E4 0,E5 0,E6 0}
   E6POS P1_K_2_App2Place={X 289.34829,Y 416.70443,Z 802.77226,A -180,B 0,C 180,S 2,T 2,E1 0,E2 0,E3 0,E4 0,E5 0,E6 0}
   E6POS P1_K_2_Place={X 289.34787,Y 316.70418,Z 652.77183,A -180,B 0,C 180,S 2,T 2,E1 0,E2 0,E3 0,E4 0,E5 0,E6 0}
   E6POS P1_K_3_App1Place={X 709.18349,Y 836.49369,Z 1002.77226,A -180,B 0,C -180,S 2,T 2,E1 0,E2 0,E3 0,E4 0,E5 0,E6 0}
   E6POS P1_K_3_App2Place={X 709.18357,Y 836.4934,Z 802.77226,A -180,B 0,C -180,S 2,T 2,E1 0,E2 0,E3 0,E4 0,E5 0,E6 0}
   E6POS P1_K_3_Place={X 709.18379,Y 736.49338,Z 652.77183,A -180,B 0,C -180,S 2,T 2,E1 0,E2 0,E3 0,E4 0,E5 0,E6 0}
   E6POS P1_K_4_App1Place={X 33.34875,Y 1092.70482,Z 1002.77226,A -180,B 0,C -180,S 2,T 2,E1 0,E2 0,E3 0,E4 0,E5 0,E6 0}
   E6POS P1_K_4_App2Place={X 33.34872,Y 1092.70456,Z 802.77226,A -180,B 0,C 180,S 2,T 18,E1 0,E2 0,E3 0,E4 0,E5 0,E6 0}
   E6POS P1_K_4_Place={X 33.34906,Y 992.70434,Z 652.77183,A -180,B 0,C -180,S 2,T 18,E1 0,E2 0,E3 0,E4 0,E5 0,E6 0}
   E6POS P1_K_5_App1Place={X 135.86633,Y -91.91463,Z 1002.77226,A 90,B 0,C 180,S 2,T 2,E1 0,E2 0,E3 0,E4 0,E5 0,E6 0}
   E6POS P1_K_5_App2Place={X 135.86633,Y -91.91463,Z 802.77226,A 90,B 0,C 180,S 2,T 2,E1 0,E2 0,E3 0,E4 0,E5 0,E6 0}
   E6POS P1_K_5_Place={X 230.11027,Y 4.30843,Z 652.77183,A 90,B 0,C 180,S 2,T 34,E1 0,E2 0,E3 0,E4 0,E5 0,E6 0}
   E6POS P1_K_6_App1Place={X 867.49529,Y 1243.09348,Z 1002.77226,A -90.00003,B 0,C 180,S 2,T 2,E1 0,E2 0,E3 0,E4 0,E5 0,E6 0}
   E6POS P1_K_6_App2Place={X 867.4955,Y 1243.0937,Z 802.77226,A -90.00001,B 0,C 180,S 2,T 18,E1 0,E2 0,E3 0,E4 0,E5 0,E6 0}
   E6POS P1_K_6_Place={X 767.4955,Y 1193.0937,Z 652.77183,A -90.00001,B 0,C 180,S 2,T 18,E1 0,E2 0,E3 0,E4 0,E5 0,E6 0}
   E6POS P1_K_7_App1Place={X 709.18357,Y 160.49357,Z 1002.77226,A -180,B 0,C 180,S 2,T 2,E1 0,E2 0,E3 0,E4 0,E5 0,E6 0}
   E6POS P1_K_7_App2Place={X 709.18356,Y 160.49366,Z 802.77226,A -180,B 0,C 180,S 2,T 2,E1 0,E2 0,E3 0,E4 0,E5 0,E6 0}
   E6POS P1_K_7_Place={X 709.18265,Y 60.49314,Z 652.77183,A -180,B 0,C 180,S 2,T 2,E1 0,E2 0,E3 0,E4 0,E5 0,E6 0}
   E6POS P1_K_8_App1Place={X 33.34862,Y 416.70458,Z 1002.77226,A -180,B 0,C 180,S 2,T 2,E1 0,E2 0,E3 0,E4 0,E5 0,E6 0}
   E6POS P1_K_8_App2Place={X 33.34863,Y 416.70468,Z 802.77226,A -180,B 0,C 180,S 2,T 2,E1 0,E2 0,E3 0,E4 0,E5 0,E6 0}
   E6POS P1_K_8_Place={X 33.3492,Y 316.7046,Z 652.77183,A -180,B 0,C -180,S 2,T 2,E1 0,E2 0,E3 0,E4 0,E5 0,E6 0}
   E6POS P1_K_9_App1Place={X 965.18393,Y 836.49268,Z 1002.77226,A -180,B 0,C 180,S 2,T 2,E1 0,E2 0,E3 0,E4 0,E5 0,E6 0}
   E6POS P1_K_9_App2Place={X 965.18406,Y 836.49238,Z 802.77226,A -180,B 0,C -180,S 2,T 2,E1 0,E2 0,E3 0,E4 0,E5 0,E6 0}
   E6POS P1_K_9_Place={X 965.18419,Y 736.49329,Z 652.77183,A -180,B 0,C 180,S 2,T 2,E1 0,E2 0,E3 0,E4 0,E5 0,E6 0}
   E6POS P1_K_10_App1Place={X 289.34895,Y 1092.70481,Z 1002.77226,A -180,B 0,C 180,S 2,T 2,E1 0,E2 0,E3 0,E4 0,E5 0,E6 0}
   E6POS P1_K_10_App2Place={X 289.34898,Y 1092.70437,Z 802.77226,A -180,B 0,C 180,S 2,T 2,E1 0,E2 0,E3 0,E4 0,E5 0,E6 0}
   E6POS P1_K_10_Place={X 289.34887,Y 992.70441,Z 652.77183,A -180,B 0,C 180,S 2,T 2,E1 0,E2 0,E3 0,E4 0,E5 0,E6 0}
   E6POS P1_K_11_App1Place={X 132.98765,Y 1243.08572,Z 1002.77226,A -90,B 0,C 180,S 2,T 2,E1 0,E2 0,E3 0,E4 0,E5 0,E6 0}
   E6POS P1_K_11_App2Place={X 132.98733,Y 1243.08625,Z 802.77226,A -90,B 0,C 180,S 2,T 2,E1 0,E2 0,E3 0,E4 0,E5 0,E6 0}
   E6POS P1_K_11_Place={X 232.98733,Y 1193.08625,Z 652.77183,A -90,B 0,C 180,S 2,T 18,E1 0,E2 0,E3 0,E4 0,E5 0,E6 0}
   E6POS P1_K_12_App1Place={X 864.59588,Y -45.6867,Z 1002.77226,A 90,B 0,C 180,S 2,T 34,E1 0,E2 0,E3 0,E4 0,E5 0,E6 0}
   E6POS P1_K_12_App2Place={X 864.59587,Y -45.68653,Z 802.77226,A 90,B 0,C 180,S 2,T 34,E1 0,E2 0,E3 0,E4 0,E5 0,E6 0}
   E6POS P1_K_12_Place={X 764.59587,Y 4.31347,Z 652.77183,A 90,B 0,C 180,S 2,T 34,E1 0,E2 0,E3 0,E4 0,E5 0,E6 0}

   ;ENDFOLD
   ;FOLD  MosaicoL_Pallet1

   E6POS P1_L_1_App1Place={X 168.0638,Y 598.29342,Z 1070.17225,A -89.99997,B 0,C 180,S 2,T 2,E1 0,E2 0,E3 0,E4 0,E5 0,E6 0}
   E6POS P1_L_1_App2Place={X 168.06418,Y 598.29353,Z 870.17216,A -89.99997,B 0,C 180,S 2,T 2,E1 0,E2 0,E3 0,E4 0,E5 0,E6 0}
   E6POS P1_L_1_Place={X 68.06526,Y 598.29341,Z 670.17152,A -90,B 0,C 180,S 2,T 2,E1 0,E2 0,E3 0,E4 0,E5 0,E6 0}
   E6POS P1_L_2_App1Place={X 432.06355,Y 598.29319,Z 1070.17225,A -89.99997,B 0,C 180,S 2,T 2,E1 0,E2 0,E3 0,E4 0,E5 0,E6 0}
   E6POS P1_L_2_App2Place={X 432.06389,Y 598.29299,Z 870.17216,A -89.99997,B 0,C 180,S 2,T 2,E1 0,E2 0,E3 0,E4 0,E5 0,E6 0}
   E6POS P1_L_2_Place={X 332.06426,Y 598.2932,Z 670.17152,A -89.99997,B 0,C 180,S 2,T 2,E1 0,E2 0,E3 0,E4 0,E5 0,E6 0}
   E6POS P1_L_3_App1Place={X 696.09636,Y 672.23863,Z 1070.17225,A -90,B 0,C 180,S 2,T 2,E1 0,E2 0,E3 0,E4 0,E5 0,E6 0}
   E6POS P1_L_3_App2Place={X 696.09645,Y 672.23864,Z 870.17216,A -90,B 0,C 180,S 2,T 2,E1 0,E2 0,E3 0,E4 0,E5 0,E6 0}
   E6POS P1_L_3_Place={X 596.09736,Y 672.23879,Z 670.17152,A -90,B 0,C 180,S 2,T 2,E1 0,E2 0,E3 0,E4 0,E5 0,E6 0}
   E6POS P1_L_4_App1Place={X 596.09735,Y 672.23874,Z 1070.17225,A -90,B 0,C 180,S 2,T 2,E1 0,E2 0,E3 0,E4 0,E5 0,E6 0}
   E6POS P1_L_4_App2Place={X 596.09692,Y 648.23875,Z 870.17216,A -90,B 0,C 180,S 2,T 2,E1 0,E2 0,E3 0,E4 0,E5 0,E6 0}
   E6POS P1_L_4_Place={X 596.09685,Y 648.23836,Z 670.17152,A -90,B 0,C 180,S 2,T 2,E1 0,E2 0,E3 0,E4 0,E5 0,E6 0}
   E6POS P1_L_5_App1Place={X 596.09692,Y 648.23875,Z 1070.17225,A -90,B 0,C 180,S 2,T 2,E1 0,E2 0,E3 0,E4 0,E5 0,E6 0}
   E6POS P1_L_5_App2Place={X 596.09676,Y 624.23876,Z 870.17216,A -90,B 0,C 180,S 2,T 2,E1 0,E2 0,E3 0,E4 0,E5 0,E6 0}
   E6POS P1_L_5_Place={X 596.09673,Y 624.23857,Z 670.17152,A -90,B 0,C 180,S 2,T 2,E1 0,E2 0,E3 0,E4 0,E5 0,E6 0}
   E6POS P1_L_6_App1Place={X 596.09676,Y 624.23876,Z 1070.17225,A -90,B 0,C 180,S 2,T 2,E1 0,E2 0,E3 0,E4 0,E5 0,E6 0}
   E6POS P1_L_6_App2Place={X 596.09655,Y 600.23828,Z 870.17216,A -90,B 0,C 180,S 2,T 2,E1 0,E2 0,E3 0,E4 0,E5 0,E6 0}
   E6POS P1_L_6_Place={X 596.09665,Y 600.23877,Z 670.17152,A -90,B 0,C 180,S 2,T 2,E1 0,E2 0,E3 0,E4 0,E5 0,E6 0}
   E6POS P1_L_7_App1Place={X 922.09597,Y 672.23817,Z 1070.17225,A -90,B 0,C 180,S 2,T 2,E1 0,E2 0,E3 0,E4 0,E5 0,E6 0}
   E6POS P1_L_7_App2Place={X 922.09645,Y 672.23879,Z 870.17216,A -90,B 0,C 180,S 2,T 2,E1 0,E2 0,E3 0,E4 0,E5 0,E6 0}
   E6POS P1_L_7_Place={X 822.09609,Y 672.23876,Z 670.17152,A -90,B 0,C 180,S 2,T 2,E1 0,E2 0,E3 0,E4 0,E5 0,E6 0}
   E6POS P1_L_8_App1Place={X 822.09616,Y 672.23897,Z 1070.17225,A -90,B 0,C 180,S 2,T 2,E1 0,E2 0,E3 0,E4 0,E5 0,E6 0}
   E6POS P1_L_8_App2Place={X 822.09694,Y 648.23821,Z 870.17216,A -90,B 0,C 180,S 2,T 2,E1 0,E2 0,E3 0,E4 0,E5 0,E6 0}
   E6POS P1_L_8_Place={X 822.0969,Y 648.23809,Z 670.17152,A -90,B 0,C 180,S 2,T 2,E1 0,E2 0,E3 0,E4 0,E5 0,E6 0}
   E6POS P1_L_9_App1Place={X 822.09694,Y 648.23821,Z 1070.17225,A -90,B 0,C 180,S 2,T 2,E1 0,E2 0,E3 0,E4 0,E5 0,E6 0}
   E6POS P1_L_9_App2Place={X 822.09613,Y 624.23895,Z 870.17216,A -90,B 0,C 180,S 2,T 2,E1 0,E2 0,E3 0,E4 0,E5 0,E6 0}
   E6POS P1_L_9_Place={X 822.09596,Y 624.23841,Z 670.17152,A -90,B 0,C 180,S 2,T 2,E1 0,E2 0,E3 0,E4 0,E5 0,E6 0}
   E6POS P1_L_10_App1Place={X 822.09613,Y 624.23895,Z 1070.17225,A -90,B 0,C 180,S 2,T 2,E1 0,E2 0,E3 0,E4 0,E5 0,E6 0}
   E6POS P1_L_10_App2Place={X 822.09631,Y 600.23873,Z 870.17216,A -90,B 0,C 180,S 2,T 2,E1 0,E2 0,E3 0,E4 0,E5 0,E6 0}
   E6POS P1_L_10_Place={X 822.09637,Y 600.23894,Z 670.17152,A -90,B 0,C 180,S 2,T 2,E1 0,E2 0,E3 0,E4 0,E5 0,E6 0}
   E6POS P1_L_11_App1Place={X 168.09579,Y 672.23859,Z 1070.17225,A -90,B 0,C 180,S 2,T 2,E1 0,E2 0,E3 0,E4 0,E5 0,E6 0}
   E6POS P1_L_11_App2Place={X 168.09611,Y 672.2387,Z 870.17216,A -90,B 0,C 180,S 2,T 2,E1 0,E2 0,E3 0,E4 0,E5 0,E6 0}
   E6POS P1_L_11_Place={X 68.09697,Y 672.23897,Z 670.17152,A -90,B 0,C 180,S 2,T 2,E1 0,E2 0,E3 0,E4 0,E5 0,E6 0}
   E6POS P1_L_12_App1Place={X 68.09697,Y 672.23896,Z 1070.17225,A -90,B 0,C 180,S 2,T 2,E1 0,E2 0,E3 0,E4 0,E5 0,E6 0}
   E6POS P1_L_12_App2Place={X 68.09599,Y 648.23858,Z 870.17216,A -90,B 0,C 180,S 2,T 2,E1 0,E2 0,E3 0,E4 0,E5 0,E6 0}
   E6POS P1_L_12_Place={X 68.09599,Y 648.23861,Z 670.17152,A -90,B 0,C 180,S 2,T 2,E1 0,E2 0,E3 0,E4 0,E5 0,E6 0}
   E6POS P1_L_13_App1Place={X 68.09599,Y 648.23858,Z 1070.17225,A -90,B 0,C 180,S 2,T 2,E1 0,E2 0,E3 0,E4 0,E5 0,E6 0}
   E6POS P1_L_13_App2Place={X 68.09686,Y 624.23871,Z 870.17216,A -90,B 0,C 180,S 2,T 2,E1 0,E2 0,E3 0,E4 0,E5 0,E6 0}
   E6POS P1_L_13_Place={X 68.09685,Y 624.23882,Z 670.17152,A -90,B 0,C 180,S 2,T 2,E1 0,E2 0,E3 0,E4 0,E5 0,E6 0}
   E6POS P1_L_14_App1Place={X 68.09686,Y 624.23871,Z 1070.17225,A -90,B 0,C 180,S 2,T 2,E1 0,E2 0,E3 0,E4 0,E5 0,E6 0}
   E6POS P1_L_14_App2Place={X 68.09658,Y 600.23864,Z 870.17216,A -90,B 0,C 180,S 2,T 2,E1 0,E2 0,E3 0,E4 0,E5 0,E6 0}
   E6POS P1_L_14_Place={X 68.09658,Y 600.2387,Z 670.17152,A -90,B 0,C 180,S 2,T 2,E1 0,E2 0,E3 0,E4 0,E5 0,E6 0}
   E6POS P1_L_15_App1Place={X 394.09588,Y 672.23849,Z 1070.17225,A -90,B 0,C 180,S 2,T 2,E1 0,E2 0,E3 0,E4 0,E5 0,E6 0}
   E6POS P1_L_15_App2Place={X 394.09624,Y 672.23892,Z 870.17216,A -90,B 0,C 180,S 2,T 2,E1 0,E2 0,E3 0,E4 0,E5 0,E6 0}
   E6POS P1_L_15_Place={X 294.09682,Y 672.23896,Z 670.17152,A -90,B 0,C 180,S 2,T 2,E1 0,E2 0,E3 0,E4 0,E5 0,E6 0}
   E6POS P1_L_16_App1Place={X 294.09682,Y 672.23888,Z 1070.17225,A -90,B 0,C 180,S 2,T 2,E1 0,E2 0,E3 0,E4 0,E5 0,E6 0}
   E6POS P1_L_16_App2Place={X 294.09703,Y 648.23826,Z 870.17216,A -90,B 0,C 180,S 2,T 2,E1 0,E2 0,E3 0,E4 0,E5 0,E6 0}
   E6POS P1_L_16_Place={X 294.09704,Y 648.23851,Z 670.17152,A -90,B 0,C 180,S 2,T 2,E1 0,E2 0,E3 0,E4 0,E5 0,E6 0}
   E6POS P1_L_17_App1Place={X 294.09703,Y 648.23826,Z 1070.17225,A -90,B 0,C 180,S 2,T 2,E1 0,E2 0,E3 0,E4 0,E5 0,E6 0}
   E6POS P1_L_17_App2Place={X 294.09602,Y 624.23846,Z 870.17216,A -90,B 0,C 180,S 2,T 2,E1 0,E2 0,E3 0,E4 0,E5 0,E6 0}
   E6POS P1_L_17_Place={X 294.09601,Y 624.23832,Z 670.17152,A -90,B 0,C 180,S 2,T 2,E1 0,E2 0,E3 0,E4 0,E5 0,E6 0}
   E6POS P1_L_18_App1Place={X 294.09602,Y 624.23846,Z 1070.17225,A -90,B 0,C 180,S 2,T 2,E1 0,E2 0,E3 0,E4 0,E5 0,E6 0}
   E6POS P1_L_18_App2Place={X 294.09608,Y 600.23829,Z 870.17216,A -90,B 0,C 180,S 2,T 2,E1 0,E2 0,E3 0,E4 0,E5 0,E6 0}
   E6POS P1_L_18_Place={X 294.0961,Y 600.23879,Z 670.17152,A -90,B 0,C 180,S 2,T 2,E1 0,E2 0,E3 0,E4 0,E5 0,E6 0}
   E6POS P1_L_19_App1Place={X 620.06456,Y 598.29327,Z 1070.17225,A -90,B 0,C 180,S 2,T 2,E1 0,E2 0,E3 0,E4 0,E5 0,E6 0}
   E6POS P1_L_19_App2Place={X 620.06428,Y 598.29308,Z 870.17216,A -90,B 0,C 180,S 2,T 2,E1 0,E2 0,E3 0,E4 0,E5 0,E6 0}
   E6POS P1_L_19_Place={X 520.06414,Y 598.29313,Z 670.17152,A -89.99997,B 0,C 180,S 2,T 2,E1 0,E2 0,E3 0,E4 0,E5 0,E6 0}
   E6POS P1_L_20_App1Place={X 884.06417,Y 598.2935,Z 1070.17225,A -89.99997,B 0,C 180,S 2,T 2,E1 0,E2 0,E3 0,E4 0,E5 0,E6 0}
   E6POS P1_L_20_App2Place={X 884.06402,Y 598.29325,Z 870.17216,A -89.99997,B 0,C 180,S 2,T 2,E1 0,E2 0,E3 0,E4 0,E5 0,E6 0}
   E6POS P1_L_20_Place={X 784.0648,Y 598.29314,Z 670.17152,A -90,B 0,C 180,S 2,T 2,E1 0,E2 0,E3 0,E4 0,E5 0,E6 0}

   ;ENDFOLD
   ;FOLD  MosaicoM_Pallet1

   E6POS P1_M_1_App1Place={X 185.75126,Y 502.65429,Z 990.17138,A -90,B 0,C 180,S 2,T 2,E1 0,E2 0,E3 0,E4 0,E5 0,E6 0}
   E6POS P1_M_1_App2Place={X 185.75082,Y 502.65481,Z 840.17071,A -90,B 0,C 180,S 2,T 2,E1 0,E2 0,E3 0,E4 0,E5 0,E6 0}
   E6POS P1_M_1_Place={X 60.91841,Y 601.45505,Z 670.17075,A -90,B 0,C 180,S 2,T 2,E1 0,E2 0,E3 0,E4 0,E5 0,E6 0}
   E6POS P1_M_2_App1Place={X 583.64064,Y 604.9628,Z 990.17138,A 90,B 0,C 180,S 2,T 34,E1 0,E2 0,E3 0,E4 0,E5 0,E6 0}
   E6POS P1_M_2_App2Place={X 583.64023,Y 604.96238,Z 840.17071,A 90,B 0,C 180,S 2,T 34,E1 0,E2 0,E3 0,E4 0,E5 0,E6 0}
   E6POS P1_M_2_Place={X 483.6401,Y 604.96221,Z 670.17075,A 90,B 0,C 180,S 2,T 34,E1 0,E2 0,E3 0,E4 0,E5 0,E6 0}
   E6POS P1_M_3_App1Place={X 969.64119,Y 604.96275,Z 990.17138,A 90,B 0,C 180,S 2,T 34,E1 0,E2 0,E3 0,E4 0,E5 0,E6 0}
   E6POS P1_M_3_App2Place={X 969.64086,Y 604.96213,Z 840.17071,A 90,B 0,C 180,S 2,T 34,E1 0,E2 0,E3 0,E4 0,E5 0,E6 0}
   E6POS P1_M_3_Place={X 869.64032,Y 604.96203,Z 670.17075,A 90,B 0,C 180,S 2,T 34,E1 0,E2 0,E3 0,E4 0,E5 0,E6 0}
   E6POS P1_M_4_App1Place={X 350.64886,Y 605.90322,Z 990.17138,A 90,B 0,C 180,S 2,T 34,E1 0,E2 0,E3 0,E4 0,E5 0,E6 0}
   E6POS P1_M_4_App2Place={X 350.64912,Y 605.90307,Z 840.17071,A 90,B 0,C 180,S 2,T 34,E1 0,E2 0,E3 0,E4 0,E5 0,E6 0}
   E6POS P1_M_4_Place={X 250.64929,Y 605.90345,Z 670.17075,A 90,B 0,C 180,S 2,T 34,E1 0,E2 0,E3 0,E4 0,E5 0,E6 0}
   E6POS P1_M_5_App1Place={X 736.64933,Y 605.90358,Z 990.17138,A 90,B 0,C 180,S 2,T 34,E1 0,E2 0,E3 0,E4 0,E5 0,E6 0}
   E6POS P1_M_5_App2Place={X 736.64908,Y 605.90347,Z 840.17071,A 90,B 0,C 180,S 2,T 34,E1 0,E2 0,E3 0,E4 0,E5 0,E6 0}
   E6POS P1_M_5_Place={X 636.64962,Y 605.90316,Z 670.17075,A 90,B 0,C 180,S 2,T 34,E1 0,E2 0,E3 0,E4 0,E5 0,E6 0}
   E6POS P1_M_6_App1Place={X 957.75126,Y 505.60746,Z 990.17138,A -90,B 0,C 180,S 2,T 2,E1 0,E2 0,E3 0,E4 0,E5 0,E6 0}
   E6POS P1_M_6_App2Place={X 957.75127,Y 505.60744,Z 840.17071,A -90,B 0,C -180,S 2,T 2,E1 0,E2 0,E3 0,E4 0,E5 0,E6 0}
   E6POS P1_M_6_Place={X 832.91967,Y 604.65501,Z 670.17075,A -90,B 0,C 180,S 2,T 2,E1 0,E2 0,E3 0,E4 0,E5 0,E6 0}

   ;ENDFOLD
   ;FOLD  MosaicoN_Pallet1

   E6POS P1_N_1_App1Place={X 133.08103,Y 567.70534,Z 953.39135,A 90,B 0,C 180,S 2,T 2,E1 0,E2 0,E3 0,E4 0,E5 0,E6 0}
   E6POS P1_N_1_App2Place={X 133.08067,Y 567.70599,Z 803.39085,A 90,B 0,C -180,S 2,T 2,E1 0,E2 0,E3 0,E4 0,E5 0,E6 0}
   E6POS P1_N_1_Place={X 83.08067,Y 567.70599,Z 653.39085,A 90,B 0,C -180,S 2,T 2,E1 0,E2 0,E3 0,E4 0,E5 0,E6 0}
   E6POS P1_N_2_App1Place={X 658.69042,Y 231.29357,Z 953.39135,A 0,B 0,C 180,S 2,T 34,E1 0,E2 0,E3 0,E4 0,E5 0,E6 0}
   E6POS P1_N_2_App2Place={X 658.69044,Y 231.29349,Z 803.39085,A 0,B 0,C -180,S 2,T 34,E1 0,E2 0,E3 0,E4 0,E5 0,E6 0}
   E6POS P1_N_2_Place={X 658.68978,Y 381.29352,Z 653.39085,A 0,B 0,C 180,S 2,T 34,E1 0,E2 0,E3 0,E4 0,E5 0,E6 0}
   E6POS P1_N_3_App1Place={X 401.08402,Y 1121.71611,Z 953.39135,A 90,B 0,C -180,S 2,T 50,E1 0,E2 0,E3 0,E4 0,E5 0,E6 0}
   E6POS P1_N_3_App2Place={X 401.08405,Y 1121.7159,Z 803.39085,A 90,B 0,C 180,S 2,T 50,E1 0,E2 0,E3 0,E4 0,E5 0,E6 0}
   E6POS P1_N_3_Place={X 301.08415,Y 1071.71593,Z 653.39085,A 90,B 0,C 180,S 2,T 50,E1 0,E2 0,E3 0,E4 0,E5 0,E6 0}
   E6POS P1_N_4_App1Place={X -97.28938,Y 63.29394,Z 953.39135,A 0,B 0,C 180,S 2,T 34,E1 0,E2 0,E3 0,E4 0,E5 0,E6 0}
   E6POS P1_N_4_App2Place={X -97.28973,Y 63.29387,Z 803.39085,A 0,B 0,C 180,S 2,T 34,E1 0,E2 0,E3 0,E4 0,E5 0,E6 0}
   E6POS P1_N_4_Place={X -97.28973,Y 163.29387,Z 653.39085,A 0,B 0,C 180,S 2,T 34,E1 0,E2 0,E3 0,E4 0,E5 0,E6 0}
   E6POS P1_N_5_App1Place={X 687.08154,Y 635.7258,Z 953.39135,A 90,B 0,C 180,S 2,T 34,E1 0,E2 0,E3 0,E4 0,E5 0,E6 0}
   E6POS P1_N_5_App2Place={X 687.08127,Y 635.72551,Z 803.39085,A 90,B 0,C 180,S 2,T 34,E1 0,E2 0,E3 0,E4 0,E5 0,E6 0}
   E6POS P1_N_5_Place={X 587.08127,Y 635.72551,Z 653.39085,A 90,B 0,C 180,S 2,T 34,E1 0,E2 0,E3 0,E4 0,E5 0,E6 0}
   E6POS P1_N_6_App1Place={X 1138.64844,Y 916.09576,Z 953.39135,A -180,B 0,C -180,S 2,T 2,E1 0,E2 0,E3 0,E4 0,E5 0,E6 0}
   E6POS P1_N_6_App2Place={X 1138.6483,Y 916.09602,Z 803.39085,A 180,B 0,C 180,S 2,T 2,E1 0,E2 0,E3 0,E4 0,E5 0,E6 0}
   E6POS P1_N_6_Place={X 1088.6483,Y 816.09602,Z 653.39085,A 180,B 0,C 180,S 2,T 2,E1 0,E2 0,E3 0,E4 0,E5 0,E6 0}
   E6POS P1_N_7_App1Place={X 905.08036,Y 81.72604,Z 953.39135,A 90,B 0,C 180,S 2,T 34,E1 0,E2 0,E3 0,E4 0,E5 0,E6 0}
   E6POS P1_N_7_App2Place={X 905.08036,Y 81.72604,Z 803.39085,A 90,B 0,C 180,S 2,T 34,E1 0,E2 0,E3 0,E4 0,E5 0,E6 0}
   E6POS P1_N_7_Place={X 805.08036,Y 131.72605,Z 653.39085,A 90,B 0,C 180,S 2,T 34,E1 0,E2 0,E3 0,E4 0,E5 0,E6 0}
   E6POS P1_N_8_App1Place={X 1188.64815,Y 1134.09646,Z 953.39135,A -180,B 0,C 180,S 2,T 2,E1 0,E2 0,E3 0,E4 0,E5 0,E6 0}
   E6POS P1_N_8_App2Place={X 1188.64815,Y 1134.09646,Z 803.39085,A -180,B 0,C 180,S 2,T 2,E1 0,E2 0,E3 0,E4 0,E5 0,E6 0}
   E6POS P1_N_8_Place={X 1088.6488,Y 1034.09614,Z 653.39085,A -180,B 0,C 180,S 2,T 2,E1 0,E2 0,E3 0,E4 0,E5 0,E6 0}

   ;ENDFOLD
   ;FOLD  MosaicoO_Pallet1

   E6POS P1_O_1_App1Place={X 935.79448,Y 172.66118,Z 845.88523,A -180,B 0,C -180,S 2,T 2,E1 0,E2 0,E3 0,E4 0,E5 0,E6 0}
   E6POS P1_O_1_App2Place={X 935.79436,Y 172.66159,Z 745.8848,A -180,B 0,C 180,S 2,T 2,E1 0,E2 0,E3 0,E4 0,E5 0,E6 0}
   E6POS P1_O_1_Place={X 935.79476,Y 72.66105,Z 645.88524,A -180,B 0,C 180,S 2,T 2,E1 0,E2 0,E3 0,E4 0,E5 0,E6 0}
   E6POS P1_O_2_App1Place={X 329.01324,Y 456.78558,Z 845.88523,A -180,B 0,C -180,S 2,T 2,E1 0,E2 0,E3 0,E4 0,E5 0,E6 0}
   E6POS P1_O_2_App2Place={X 329.01325,Y 456.7853,Z 745.8848,A -180,B 0,C 180,S 2,T 2,E1 0,E2 0,E3 0,E4 0,E5 0,E6 0}
   E6POS P1_O_2_Place={X 329.01323,Y 356.78607,Z 645.88524,A -180,B 0,C 180,S 2,T 2,E1 0,E2 0,E3 0,E4 0,E5 0,E6 0}
   E6POS P1_O_3_App1Place={X 651.79561,Y 780.66165,Z 845.88523,A -180,B 0,C 180,S 2,T 2,E1 0,E2 0,E3 0,E4 0,E5 0,E6 0}
   E6POS P1_O_3_App2Place={X 651.79565,Y 780.6615,Z 745.8848,A -180,B 0,C -180,S 2,T 2,E1 0,E2 0,E3 0,E4 0,E5 0,E6 0}
   E6POS P1_O_3_Place={X 651.79572,Y 680.66131,Z 645.88524,A -180,B 0,C 180,S 2,T 2,E1 0,E2 0,E3 0,E4 0,E5 0,E6 0}
   E6POS P1_O_4_App1Place={X 45.01229,Y 1064.78633,Z 845.88523,A -180,B 0,C 180,S 2,T 18,E1 0,E2 0,E3 0,E4 0,E5 0,E6 0}
   E6POS P1_O_4_App2Place={X 45.01228,Y 1064.78624,Z 745.8848,A -180,B 0,C 180,S 2,T 18,E1 0,E2 0,E3 0,E4 0,E5 0,E6 0}
   E6POS P1_O_4_Place={X 45.01235,Y 964.78626,Z 645.88524,A -180,B 0,C 180,S 2,T 18,E1 0,E2 0,E3 0,E4 0,E5 0,E6 0}
   E6POS P1_O_5_App1Place={X 170.85014,Y -87.51639,Z 845.88523,A 90,B 0,C 180,S 2,T 2,E1 0,E2 0,E3 0,E4 0,E5 0,E6 0}
   E6POS P1_O_5_App2Place={X 170.85014,Y -87.51635,Z 745.8848,A 90,B 0,C 180,S 2,T 2,E1 0,E2 0,E3 0,E4 0,E5 0,E6 0}
   E6POS P1_O_5_Place={X 270.85006,Y 12.48387,Z 645.88524,A 90,B 0,C 180,S 2,T 34,E1 0,E2 0,E3 0,E4 0,E5 0,E6 0}
   E6POS P1_O_6_App1Place={X 828.97521,Y 1287.2666,Z 845.88523,A -90,B 0,C -180,S 2,T 18,E1 0,E2 0,E3 0,E4 0,E5 0,E6 0}
   E6POS P1_O_6_App2Place={X 828.97552,Y 1287.26658,Z 745.8848,A -90,B 0,C 180,S 2,T 18,E1 0,E2 0,E3 0,E4 0,E5 0,E6 0}
   E6POS P1_O_6_Place={X 714.4457,Y 1187.27407,Z 645.88524,A -90,B 0,C 180,S 2,T 18,E1 0,E2 0,E3 0,E4 0,E5 0,E6 0}
   E6POS P1_O_7_App1Place={X 651.79639,Y 172.66167,Z 845.88523,A -180,B 0,C -180,S 2,T 2,E1 0,E2 0,E3 0,E4 0,E5 0,E6 0}
   E6POS P1_O_7_App2Place={X 651.79644,Y 172.6614,Z 745.8848,A -180,B 0,C 180,S 2,T 2,E1 0,E2 0,E3 0,E4 0,E5 0,E6 0}
   E6POS P1_O_7_Place={X 651.79621,Y 72.66195,Z 645.88524,A -180,B 0,C 180,S 2,T 2,E1 0,E2 0,E3 0,E4 0,E5 0,E6 0}
   E6POS P1_O_8_App1Place={X 45.01296,Y 456.78658,Z 845.88523,A -180,B 0,C -180,S 2,T 2,E1 0,E2 0,E3 0,E4 0,E5 0,E6 0}
   E6POS P1_O_8_App2Place={X 45.01296,Y 456.78657,Z 745.8848,A -180,B 0,C 180,S 2,T 2,E1 0,E2 0,E3 0,E4 0,E5 0,E6 0}
   E6POS P1_O_8_Place={X 45.0129,Y 356.78655,Z 645.88524,A -180,B 0,C 180,S 2,T 2,E1 0,E2 0,E3 0,E4 0,E5 0,E6 0}
   E6POS P1_O_9_App1Place={X 935.79619,Y 780.66198,Z 845.88523,A 180,B 0,C -180,S 2,T 2,E1 0,E2 0,E3 0,E4 0,E5 0,E6 0}
   E6POS P1_O_9_App2Place={X 935.79625,Y 780.66184,Z 745.8848,A -180,B 0,C -180,S 2,T 2,E1 0,E2 0,E3 0,E4 0,E5 0,E6 0}
   E6POS P1_O_9_Place={X 935.79614,Y 680.66184,Z 645.88524,A -180,B 0,C 180,S 2,T 2,E1 0,E2 0,E3 0,E4 0,E5 0,E6 0}
   E6POS P1_O_10_App1Place={X 329.01319,Y 1064.7858,Z 845.88523,A 180,B 0,C -180,S 2,T 2,E1 0,E2 0,E3 0,E4 0,E5 0,E6 0}
   E6POS P1_O_10_App2Place={X 329.0132,Y 1064.78566,Z 745.8848,A -180,B 0,C 180,S 2,T 2,E1 0,E2 0,E3 0,E4 0,E5 0,E6 0}
   E6POS P1_O_10_Place={X 329.01301,Y 964.78561,Z 645.88524,A -180,B 0,C -180,S 2,T 18,E1 0,E2 0,E3 0,E4 0,E5 0,E6 0}
   E6POS P1_O_11_App1Place={X 878.85065,Y -37.51507,Z 845.88523,A 90,B 0,C 180,S 2,T 34,E1 0,E2 0,E3 0,E4 0,E5 0,E6 0}
   E6POS P1_O_11_App2Place={X 878.85073,Y -37.51535,Z 745.8848,A 90,B 0,C 180,S 2,T 34,E1 0,E2 0,E3 0,E4 0,E5 0,E6 0}
   E6POS P1_O_11_Place={X 713.184,Y 15.84173,Z 645.88524,A 90,B 0,C 180,S 2,T 34,E1 0,E2 0,E3 0,E4 0,E5 0,E6 0}
   E6POS P1_O_12_App1Place={X 170.97564,Y 1287.2668,Z 845.88523,A -90,B 0,C 180,S 2,T 18,E1 0,E2 0,E3 0,E4 0,E5 0,E6 0}
   E6POS P1_O_12_App2Place={X 170.97564,Y 1287.26676,Z 745.8848,A -90,B 0,C 180,S 2,T 18,E1 0,E2 0,E3 0,E4 0,E5 0,E6 0}
   E6POS P1_O_12_Place={X 270.97608,Y 1187.26674,Z 645.88524,A -90,B 0,C 180,S 2,T 18,E1 0,E2 0,E3 0,E4 0,E5 0,E6 0}

   ;ENDFOLD
   ;FOLD  MosaicoP1_Pallet1

   E6POS P1_P_1_App1Place={X 617.07431,Y 364.14311,Z 890.16691,A -180,B 0,C -180,S 2,T 2,E1 0,E2 0,E3 0,E4 0,E5 0,E6 0}
   E6POS P1_P_1_App2Place={X 617.07384,Y 364.14354,Z 740.16729,A -180,B 0,C 180,S 2,T 2,E1 0,E2 0,E3 0,E4 0,E5 0,E6 0}
   E6POS P1_P_1_Place={X 616.25932,Y 251.52907,Z 660.09943,A -180,B 0,C 180,S 2,T 2,E1 0,E2 0,E3 0,E4 0,E5 0,E6 0}
   E6POS P1_P_2_App1Place={X 17.29738,Y 778.4879,Z 890.16691,A -180,B 0,C -180,S 2,T 2,E1 0,E2 0,E3 0,E4 0,E5 0,E6 0}
   E6POS P1_P_2_App2Place={X 17.2976,Y 778.48775,Z 740.16729,A -180,B 0,C 180,S 2,T 2,E1 0,E2 0,E3 0,E4 0,E5 0,E6 0}
   E6POS P1_P_2_Place={X 17.29771,Y 665.87327,Z 660.09943,A -180,B 0,C 180,S 2,T 2,E1 0,E2 0,E3 0,E4 0,E5 0,E6 0}
   E6POS P1_P_3_App1Place={X 616.25934,Y 1194.14061,Z 890.16691,A -180,B 0,C -180,S 2,T 18,E1 0,E2 0,E3 0,E4 0,E5 0,E6 0}
   E6POS P1_P_3_App2Place={X 616.25968,Y 1194.1408,Z 740.16729,A -180,B 0,C 180,S 2,T 18,E1 0,E2 0,E3 0,E4 0,E5 0,E6 0}
   E6POS P1_P_3_Place={X 616.25957,Y 1081.52903,Z 660.09943,A -180,B 0,C -180,S 2,T 18,E1 0,E2 0,E3 0,E4 0,E5 0,E6 0}
   E6POS P1_P_4_App1Place={X 1099.03595,Y 595.11583,Z 890.16691,A 90,B 0,C 180,S 2,T 34,E1 0,E2 0,E3 0,E4 0,E5 0,E6 0}
   E6POS P1_P_4_App2Place={X 1099.03552,Y 595.11554,Z 740.16729,A 90,B 0,C 180,S 2,T 34,E1 0,E2 0,E3 0,E4 0,E5 0,E6 0}
   E6POS P1_P_4_Place={X 875.78418,Y 595.11547,Z 660.09943,A 90,B 0,C 180,S 2,T 34,E1 0,E2 0,E3 0,E4 0,E5 0,E6 0}
   E6POS P1_P_5_App1Place={X 986.25997,Y 364.13451,Z 890.16691,A -180,B 0,C 180,S 2,T 2,E1 0,E2 0,E3 0,E4 0,E5 0,E6 0}
   E6POS P1_P_5_App2Place={X 986.25979,Y 364.13425,Z 740.16729,A -180,B 0,C 180,S 2,T 2,E1 0,E2 0,E3 0,E4 0,E5 0,E6 0}
   E6POS P1_P_5_Place={X 986.25884,Y 251.548,Z 660.09943,A -180,B 0,C 180,S 2,T 2,E1 0,E2 0,E3 0,E4 0,E5 0,E6 0}
   E6POS P1_P_6_App1Place={X 387.29652,Y 778.47742,Z 890.16691,A -180,B 0,C 180,S 2,T 2,E1 0,E2 0,E3 0,E4 0,E5 0,E6 0}
   E6POS P1_P_6_App2Place={X 387.29629,Y 778.47753,Z 740.16729,A -180,B 0,C 180,S 2,T 2,E1 0,E2 0,E3 0,E4 0,E5 0,E6 0}
   E6POS P1_P_6_Place={X 387.29686,Y 665.89221,Z 660.09943,A -180,B 0,C 180,S 2,T 2,E1 0,E2 0,E3 0,E4 0,E5 0,E6 0}
   E6POS P1_P_7_App1Place={X 986.25937,Y 1194.13488,Z 890.16691,A -180,B 0,C -180,S 2,T 2,E1 0,E2 0,E3 0,E4 0,E5 0,E6 0}
   E6POS P1_P_7_App2Place={X 986.25917,Y 1194.13486,Z 740.16729,A -180,B 0,C 180,S 2,T 2,E1 0,E2 0,E3 0,E4 0,E5 0,E6 0}
   E6POS P1_P_7_Place={X 986.25895,Y 1081.54783,Z 660.09943,A -180,B 0,C 180,S 2,T 2,E1 0,E2 0,E3 0,E4 0,E5 0,E6 0}
   E6POS P1_P_8_App1Place={X 45.93133,Y 593.04257,Z 890.16691,A -90,B 0,C 180,S 2,T 2,E1 0,E2 0,E3 0,E4 0,E5 0,E6 0}
   E6POS P1_P_8_App2Place={X 45.93167,Y 593.04221,Z 740.16729,A -90,B 0,C 180,S 2,T 2,E1 0,E2 0,E3 0,E4 0,E5 0,E6 0}
   E6POS P1_P_8_Place={X 130.48397,Y 593.04207,Z 660.09943,A -90,B 0,C 180,S 2,T 2,E1 0,E2 0,E3 0,E4 0,E5 0,E6 0}

   ;ENDFOLD
   ;FOLD  MosaicoQ_Pallet1

   E6POS P1_Q_1_App1Place={X 457.55562,Y 375.4155,Z 1111.95716,A 180,B 0,C 180,S 2,T 2,E1 0,E2 0,E3 0,E4 0,E5 0,E6 0}
   E6POS P1_Q_1_App2Place={X 457.55558,Y 375.41581,Z 911.95694,A -180,B 0,C -180,S 2,T 2,E1 0,E2 0,E3 0,E4 0,E5 0,E6 0}
   E6POS P1_Q_1_Place={X 457.5548,Y 275.41596,Z 661.95611,A -180,B 0,C 180,S 2,T 2,E1 0,E2 0,E3 0,E4 0,E5 0,E6 0}
   E6POS P1_Q_2_App1Place={X 558.55606,Y 1099.41654,Z 1111.95716,A -180,B 0,C -180,S 2,T 2,E1 0,E2 0,E3 0,E4 0,E5 0,E6 0}
   E6POS P1_Q_2_App2Place={X 558.55601,Y 1099.41679,Z 911.95694,A -180,B 0,C 180,S 2,T 18,E1 0,E2 0,E3 0,E4 0,E5 0,E6 0}
   E6POS P1_Q_2_Place={X 558.55592,Y 999.41595,Z 661.95611,A -180,B 0,C 180,S 2,T 18,E1 0,E2 0,E3 0,E4 0,E5 0,E6 0}
   E6POS P1_Q_3_App1Place={X 936.32742,Y 1166.50741,Z 1111.95716,A -90,B 0,C -180,S 2,T 2,E1 0,E2 0,E3 0,E4 0,E5 0,E6 0}
   E6POS P1_Q_3_App2Place={X 936.32726,Y 1166.50773,Z 911.95694,A -90,B 0,C 180,S 2,T 2,E1 0,E2 0,E3 0,E4 0,E5 0,E6 0}
   E6POS P1_Q_3_Place={X 836.32776,Y 1066.50753,Z 661.95611,A -90,B 0,C -180,S 2,T 18,E1 0,E2 0,E3 0,E4 0,E5 0,E6 0}
   E6POS P1_Q_4_App1Place={X 40.56901,Y 30.4136,Z 1111.95716,A 90,B 0,C -180,S 2,T 2,E1 0,E2 0,E3 0,E4 0,E5 0,E6 0}
   E6POS P1_Q_4_App2Place={X 40.56901,Y 30.41346,Z 911.95694,A 90,B 0,C 180,S 2,T 2,E1 0,E2 0,E3 0,E4 0,E5 0,E6 0}
   E6POS P1_Q_4_Place={X 140.56858,Y 130.41377,Z 661.95611,A 90,B 0,C 180,S 2,T 2,E1 0,E2 0,E3 0,E4 0,E5 0,E6 0}

   ;ENDFOLD
   ;FOLD  MosaicoR_Pallet1

   E6POS P1_R_1_App1Place={X 899.62689,Y 611.46532,Z 1052.81504,A -90,B 0,C -180,S 2,T 2,E1 0,E2 0,E3 0,E4 0,E5 0,E6 0}
   E6POS P1_R_1_App2Place={X 899.62683,Y 611.4655,Z 852.81474,A -90,B 0,C 180,S 2,T 2,E1 0,E2 0,E3 0,E4 0,E5 0,E6 0}
   E6POS P1_R_1_Place={X 899.62697,Y 561.46554,Z 652.81447,A -90,B 0,C 180,S 2,T 2,E1 0,E2 0,E3 0,E4 0,E5 0,E6 0}
   E6POS P1_R_2_App1Place={X 455.62662,Y 147.46542,Z 1052.81504,A -90,B 0,C -180,S 2,T 2,E1 0,E2 0,E3 0,E4 0,E5 0,E6 0}
   E6POS P1_R_2_App2Place={X 455.62664,Y 147.46525,Z 852.81474,A -90,B 0,C 180,S 2,T 2,E1 0,E2 0,E3 0,E4 0,E5 0,E6 0}
   E6POS P1_R_2_Place={X 555.62602,Y 97.46514,Z 652.81447,A -90,B 0,C 180,S 2,T 2,E1 0,E2 0,E3 0,E4 0,E5 0,E6 0}
   E6POS P1_R_3_App1Place={X 726.31135,Y 877.74518,Z 1052.81504,A 180,B 0,C -180,S 2,T 2,E1 0,E2 0,E3 0,E4 0,E5 0,E6 0}
   E6POS P1_R_3_App2Place={X 726.31138,Y 877.74506,Z 852.81474,A -180,B 0,C 180,S 2,T 2,E1 0,E2 0,E3 0,E4 0,E5 0,E6 0}
   E6POS P1_R_3_Place={X 726.31131,Y 777.74518,Z 652.81447,A -180,B 0,C -180,S 2,T 2,E1 0,E2 0,E3 0,E4 0,E5 0,E6 0}
   E6POS P1_R_4_App1Place={X 38.31116,Y 1109.74505,Z 1052.81504,A -180,B 0,C -180,S 2,T 2,E1 0,E2 0,E3 0,E4 0,E5 0,E6 0}
   E6POS P1_R_4_App2Place={X 38.31117,Y 1109.74517,Z 852.81474,A -180,B 0,C -180,S 2,T 18,E1 0,E2 0,E3 0,E4 0,E5 0,E6 0}
   E6POS P1_R_4_Place={X 38.31156,Y 1009.7447,Z 652.81447,A -180,B 0,C 180,S 2,T 18,E1 0,E2 0,E3 0,E4 0,E5 0,E6 0}
   E6POS P1_R_5_App1Place={X 887.91772,Y 1249.24739,Z 1052.81504,A -90,B 0,C 180,S 2,T 2,E1 0,E2 0,E3 0,E4 0,E5 0,E6 0}
   E6POS P1_R_5_App2Place={X 887.9177,Y 1249.24742,Z 852.81474,A -90,B 0,C 180,S 2,T 18,E1 0,E2 0,E3 0,E4 0,E5 0,E6 0}
   E6POS P1_R_5_Place={X 787.91718,Y 1179.24698,Z 652.81447,A -90,B 0,C 180,S 2,T 18,E1 0,E2 0,E3 0,E4 0,E5 0,E6 0}
   E6POS P1_R_6_App1Place={X 153.87899,Y -80.39794,Z 1052.81504,A 90,B 0,C 180,S 2,T 2,E1 0,E2 0,E3 0,E4 0,E5 0,E6 0}
   E6POS P1_R_6_App2Place={X 153.8784,Y -80.39794,Z 852.81474,A 90,B 0,C 180,S 2,T 2,E1 0,E2 0,E3 0,E4 0,E5 0,E6 0}
   E6POS P1_R_6_Place={X 203.8784,Y 19.60206,Z 652.81447,A 90,B 0,C 180,S 2,T 34,E1 0,E2 0,E3 0,E4 0,E5 0,E6 0}
   E6POS P1_R_7_App1Place={X 899.62853,Y 1307.12146,Z 1052.81504,A -90,B 0,C 180,S 2,T 2,E1 0,E2 0,E3 0,E4 0,E5 0,E6 0}
   E6POS P1_R_7_App2Place={X 899.62822,Y 1307.12121,Z 852.81474,A -90,B 0,C 180,S 2,T 2,E1 0,E2 0,E3 0,E4 0,E5 0,E6 0}
   E6POS P1_R_7_Place={X 899.62822,Y 1257.12121,Z 652.81447,A -90,B 0,C 180,S 2,T 2,E1 0,E2 0,E3 0,E4 0,E5 0,E6 0}
   E6POS P1_R_8_App1Place={X 455.6273,Y 561.12128,Z 1052.81504,A -90,B 0,C 180,S 2,T 2,E1 0,E2 0,E3 0,E4 0,E5 0,E6 0}
   E6POS P1_R_8_App2Place={X 455.62748,Y 561.12122,Z 852.81474,A -90,B 0,C 180,S 2,T 2,E1 0,E2 0,E3 0,E4 0,E5 0,E6 0}
   E6POS P1_R_8_Place={X 555.62748,Y 561.12122,Z 652.81447,A -90,B 0,C 180,S 2,T 2,E1 0,E2 0,E3 0,E4 0,E5 0,E6 0}
   E6POS P1_R_9_App1Place={X 725.42733,Y 321.99978,Z 1052.81504,A 180,B 0,C 180,S 2,T 2,E1 0,E2 0,E3 0,E4 0,E5 0,E6 0}
   E6POS P1_R_9_App2Place={X 725.42713,Y 321.99976,Z 852.81474,A 180,B 0,C 180,S 2,T 2,E1 0,E2 0,E3 0,E4 0,E5 0,E6 0}
   E6POS P1_R_9_Place={X 725.42713,Y 421.99976,Z 652.81447,A 180,B 0,C 180,S 2,T 2,E1 0,E2 0,E3 0,E4 0,E5 0,E6 0}
   E6POS P1_R_10_App1Place={X 37.43585,Y 89.98564,Z 1052.81504,A -180,B 0,C 180,S 2,T 2,E1 0,E2 0,E3 0,E4 0,E5 0,E6 0}
   E6POS P1_R_10_App2Place={X 37.436,Y 89.98561,Z 852.81474,A 180,B 0,C 180,S 2,T 2,E1 0,E2 0,E3 0,E4 0,E5 0,E6 0}
   E6POS P1_R_10_Place={X 37.436,Y 189.98561,Z 652.81447,A 180,B 0,C 180,S 2,T 2,E1 0,E2 0,E3 0,E4 0,E5 0,E6 0}
   E6POS P1_R_11_App1Place={X 157.81215,Y 1230.13255,Z 1052.81504,A -90,B 0,C 180,S 2,T 2,E1 0,E2 0,E3 0,E4 0,E5 0,E6 0}
   E6POS P1_R_11_App2Place={X 157.81214,Y 1230.1328,Z 852.81474,A -90.00001,B 0,C 180,S 2,T 2,E1 0,E2 0,E3 0,E4 0,E5 0,E6 0}
   E6POS P1_R_11_Place={X 207.81214,Y 1180.1328,Z 652.81447,A -90.00001,B 0,C 180,S 2,T 2,E1 0,E2 0,E3 0,E4 0,E5 0,E6 0}
   E6POS P1_R_12_App1Place={X 837.91668,Y -30.40426,Z 1052.81504,A 90,B 0,C 180,S 2,T 34,E1 0,E2 0,E3 0,E4 0,E5 0,E6 0}
   E6POS P1_R_12_App2Place={X 837.91671,Y -30.40437,Z 852.81474,A 90,B 0,C 180,S 2,T 34,E1 0,E2 0,E3 0,E4 0,E5 0,E6 0}
   E6POS P1_R_12_Place={X 787.91779,Y 19.59586,Z 652.81447,A 90,B 0,C 180,S 2,T 34,E1 0,E2 0,E3 0,E4 0,E5 0,E6 0}

   ;ENDFOLD
   ;FOLD  MosaicoS_Pallet1

   E6POS P1_S_1_App1Place={X 741.07867,Y 636.24237,Z 1090.17083,A -89.99997,B 0,C 180,S 2,T 2,E1 0,E2 0,E3 0,E4 0,E5 0,E6 0}
   E6POS P1_S_1_App2Place={X 741.07843,Y 636.24271,Z 890.17129,A -89.99997,B 0,C 180,S 2,T 2,E1 0,E2 0,E3 0,E4 0,E5 0,E6 0}
   E6POS P1_S_1_Place={X 910.50314,Y 581.88157,Z 662.05452,A -89.99997,B 0,C 180,S 2,T 2,E1 0,E2 0,E3 0,E4 0,E5 0,E6 0}
   E6POS P1_S_2_App1Place={X 418.07891,Y 636.74239,Z 1090.17083,A -90,B 0,C 180,S 2,T 2,E1 0,E2 0,E3 0,E4 0,E5 0,E6 0}
   E6POS P1_S_2_App2Place={X 418.07876,Y 636.74273,Z 890.17129,A -90,B 0,C 180,S 2,T 2,E1 0,E2 0,E3 0,E4 0,E5 0,E6 0}
   E6POS P1_S_2_Place={X 587.50395,Y 582.38133,Z 662.05452,A -90,B 0,C 180,S 2,T 2,E1 0,E2 0,E3 0,E4 0,E5 0,E6 0}
   E6POS P1_S_3_App1Place={X 163.70702,Y 108.33185,Z 1090.17083,A -90,B 0,C 180,S 2,T 2,E1 0,E2 0,E3 0,E4 0,E5 0,E6 0}
   E6POS P1_S_3_App2Place={X 163.70752,Y 108.33171,Z 890.17129,A -90,B 0,C -180,S 2,T 2,E1 0,E2 0,E3 0,E4 0,E5 0,E6 0}
   E6POS P1_S_3_Place={X 263.70752,Y 108.33171,Z 662.05452,A -90,B 0,C -180,S 2,T 2,E1 0,E2 0,E3 0,E4 0,E5 0,E6 0}
   E6POS P1_S_4_App1Place={X 548.98255,Y 698.88729,Z 1090.17083,A -180,B 0,C 180,S 2,T 2,E1 0,E2 0,E3 0,E4 0,E5 0,E6 0}
   E6POS P1_S_4_App2Place={X 548.98283,Y 698.88748,Z 890.17129,A -180,B 0,C 180,S 2,T 2,E1 0,E2 0,E3 0,E4 0,E5 0,E6 0}
   E6POS P1_S_4_Place={X 548.98171,Y 596.91087,Z 662.05452,A -180,B 0,C 180,S 2,T 2,E1 0,E2 0,E3 0,E4 0,E5 0,E6 0}
   E6POS P1_S_5_App1Place={X 548.98164,Y 1001.88701,Z 1090.17083,A -180,B 0,C 180,S 2,T 2,E1 0,E2 0,E3 0,E4 0,E5 0,E6 0}
   E6POS P1_S_5_App2Place={X 548.98207,Y 1001.88729,Z 890.17129,A -180,B 0,C 180,S 2,T 2,E1 0,E2 0,E3 0,E4 0,E5 0,E6 0}
   E6POS P1_S_5_Place={X 548.98218,Y 899.91031,Z 662.05452,A -180,B 0,C -180,S 2,T 18,E1 0,E2 0,E3 0,E4 0,E5 0,E6 0}
   E6POS P1_S_6_App1Place={X 212.99271,Y 614.54265,Z 1090.17083,A 90,B 0,C 180,S 2,T 34,E1 0,E2 0,E3 0,E4 0,E5 0,E6 0}
   E6POS P1_S_6_App2Place={X 212.99282,Y 614.54256,Z 890.17129,A 90,B 0,C 180,S 2,T 34,E1 0,E2 0,E3 0,E4 0,E5 0,E6 0}
   E6POS P1_S_6_Place={X 88.77457,Y 614.54268,Z 662.05452,A 90,B 0,C 180,S 2,T 2,E1 0,E2 0,E3 0,E4 0,E5 0,E6 0}
   E6POS P1_S_7_App1Place={X 535.99323,Y 614.14252,Z 1090.17083,A 90,B 0,C 180,S 2,T 34,E1 0,E2 0,E3 0,E4 0,E5 0,E6 0}
   E6POS P1_S_7_App2Place={X 535.99309,Y 614.14264,Z 890.17129,A 90,B 0,C 180,S 2,T 34,E1 0,E2 0,E3 0,E4 0,E5 0,E6 0}
   E6POS P1_S_7_Place={X 411.77415,Y 614.14281,Z 662.05452,A 90,B 0,C 180,S 2,T 34,E1 0,E2 0,E3 0,E4 0,E5 0,E6 0}
   E6POS P1_S_8_App1Place={X 834.59202,Y 1088.58932,Z 1090.17083,A 90,B 0,C 180,S 2,T 34,E1 0,E2 0,E3 0,E4 0,E5 0,E6 0}
   E6POS P1_S_8_App2Place={X 834.59246,Y 1088.58903,Z 890.17129,A 90,B 0,C 180,S 2,T 34,E1 0,E2 0,E3 0,E4 0,E5 0,E6 0}
   E6POS P1_S_8_Place={X 734.59246,Y 1088.58903,Z 662.05452,A 90,B 0,C 180,S 2,T 34,E1 0,E2 0,E3 0,E4 0,E5 0,E6 0}
   E6POS P1_S_9_App1Place={X 449.28094,Y 499.55088,Z 1090.17083,A 0,B 0,C 180,S 2,T 34,E1 0,E2 0,E3 0,E4 0,E5 0,E6 0}
   E6POS P1_S_9_App2Place={X 449.28084,Y 499.55095,Z 890.17129,A 0,B 0,C -180,S 2,T 34,E1 0,E2 0,E3 0,E4 0,E5 0,E6 0}
   E6POS P1_S_9_Place={X 449.28092,Y 599.55096,Z 662.05452,A 0,B 0,C 180,S 2,T 34,E1 0,E2 0,E3 0,E4 0,E5 0,E6 0}
   E6POS P1_S_10_App1Place={X 449.28498,Y 196.5437,Z 1090.17083,A 0,B 0,C 180,S 2,T 34,E1 0,E2 0,E3 0,E4 0,E5 0,E6 0}
   E6POS P1_S_10_App2Place={X 449.28452,Y 196.54376,Z 890.17129,A 0,B 0,C -180,S 2,T 34,E1 0,E2 0,E3 0,E4 0,E5 0,E6 0}
   E6POS P1_S_10_Place={X 449.285,Y 296.54355,Z 662.05452,A 0,B 0,C 180,S 2,T 34,E1 0,E2 0,E3 0,E4 0,E5 0,E6 0}

   ;ENDFOLD
   ;FOLD  MosaicoT_Pallet1

   E6POS P1_T_1_App1Place={X 519.66451,Y 1058.50252,Z 970.17229,A -180,B 0,C 180,S 2,T 2,E1 0,E2 0,E3 0,E4 0,E5 0,E6 0}
   E6POS P1_T_1_App2Place={X 519.66406,Y 1058.50233,Z 820.17205,A 180,B 0,C 180,S 2,T 18,E1 0,E2 0,E3 0,E4 0,E5 0,E6 0}
   E6POS P1_T_1_Place={X 519.66406,Y 1108.50233,Z 670.17205,A 180,B 0,C 180,S 2,T 18,E1 0,E2 0,E3 0,E4 0,E5 0,E6 0}
   E6POS P1_T_2_App1Place={X 519.66406,Y 1108.50233,Z 970.17229,A 180,B 0,C 180,S 2,T 18,E1 0,E2 0,E3 0,E4 0,E5 0,E6 0}
   E6POS P1_T_2_App2Place={X 550.66406,Y 1108.50233,Z 820.17205,A 180,B 0,C 180,S 2,T 18,E1 0,E2 0,E3 0,E4 0,E5 0,E6 0}
   E6POS P1_T_2_Place={X 550.66406,Y 1108.50233,Z 670.17205,A 180,B 0,C 180,S 2,T 18,E1 0,E2 0,E3 0,E4 0,E5 0,E6 0}
   E6POS P1_T_3_App1Place={X 550.66406,Y 1108.50233,Z 970.17229,A 180,B 0,C 180,S 2,T 18,E1 0,E2 0,E3 0,E4 0,E5 0,E6 0}
   E6POS P1_T_3_App2Place={X 581.66406,Y 1108.50233,Z 820.17205,A 180,B 0,C 180,S 2,T 18,E1 0,E2 0,E3 0,E4 0,E5 0,E6 0}
   E6POS P1_T_3_Place={X 581.66406,Y 1108.50233,Z 670.17205,A 180,B 0,C 180,S 2,T 18,E1 0,E2 0,E3 0,E4 0,E5 0,E6 0}
   E6POS P1_T_4_App1Place={X 519.68036,Y 803.68304,Z 970.17229,A -180,B 0,C -180,S 2,T 2,E1 0,E2 0,E3 0,E4 0,E5 0,E6 0}
   E6POS P1_T_4_App2Place={X 519.68029,Y 803.68307,Z 820.17205,A 180,B 0,C 180,S 2,T 2,E1 0,E2 0,E3 0,E4 0,E5 0,E6 0}
   E6POS P1_T_4_Place={X 519.68029,Y 903.68307,Z 670.17205,A 180,B 0,C -180,S 2,T 18,E1 0,E2 0,E3 0,E4 0,E5 0,E6 0}
   E6POS P1_T_5_App1Place={X 519.68043,Y 490.68346,Z 970.17229,A -180,B 0,C 180,S 2,T 2,E1 0,E2 0,E3 0,E4 0,E5 0,E6 0}
   E6POS P1_T_5_App2Place={X 519.68029,Y 490.68307,Z 820.17205,A 180,B 0,C 180,S 2,T 2,E1 0,E2 0,E3 0,E4 0,E5 0,E6 0}
   E6POS P1_T_5_Place={X 519.68031,Y 590.68319,Z 670.17205,A 180,B 0,C 180,S 2,T 2,E1 0,E2 0,E3 0,E4 0,E5 0,E6 0}
   E6POS P1_T_6_App1Place={X 519.68039,Y 177.6827,Z 970.17229,A -180,B 0,C 180,S 2,T 2,E1 0,E2 0,E3 0,E4 0,E5 0,E6 0}
   E6POS P1_T_6_App2Place={X 519.68029,Y 177.68307,Z 820.17205,A 180,B 0,C 180,S 2,T 2,E1 0,E2 0,E3 0,E4 0,E5 0,E6 0}
   E6POS P1_T_6_Place={X 519.68029,Y 277.68303,Z 670.17205,A 180,B 0,C 180,S 2,T 2,E1 0,E2 0,E3 0,E4 0,E5 0,E6 0}
   E6POS P1_T_7_App1Place={X 519.68014,Y 1003.68275,Z 970.17229,A -180,B 0,C -180,S 2,T 2,E1 0,E2 0,E3 0,E4 0,E5 0,E6 0}
   E6POS P1_T_7_App2Place={X 519.68029,Y 1003.68307,Z 820.17205,A 180,B 0,C 180,S 2,T 2,E1 0,E2 0,E3 0,E4 0,E5 0,E6 0}
   E6POS P1_T_7_Place={X 519.68029,Y 1103.68303,Z 670.17205,A 180,B 0,C 180,S 2,T 18,E1 0,E2 0,E3 0,E4 0,E5 0,E6 0}
   E6POS P1_T_8_App1Place={X 519.68029,Y 690.68274,Z 970.17229,A -180,B 0,C -180,S 2,T 2,E1 0,E2 0,E3 0,E4 0,E5 0,E6 0}
   E6POS P1_T_8_App2Place={X 519.68029,Y 690.68307,Z 820.17205,A 180,B 0,C 180,S 2,T 2,E1 0,E2 0,E3 0,E4 0,E5 0,E6 0}
   E6POS P1_T_8_Place={X 519.68029,Y 790.68303,Z 670.17205,A 180,B 0,C 180,S 2,T 2,E1 0,E2 0,E3 0,E4 0,E5 0,E6 0}
   E6POS P1_T_9_App1Place={X 519.68116,Y 377.68288,Z 970.17229,A -180,B 0,C -180,S 2,T 2,E1 0,E2 0,E3 0,E4 0,E5 0,E6 0}
   E6POS P1_T_9_App2Place={X 519.68029,Y 377.68307,Z 820.17205,A 180,B 0,C 180,S 2,T 2,E1 0,E2 0,E3 0,E4 0,E5 0,E6 0}
   E6POS P1_T_9_Place={X 519.68029,Y 477.68303,Z 670.17205,A 180,B 0,C 180,S 2,T 2,E1 0,E2 0,E3 0,E4 0,E5 0,E6 0}
   E6POS P1_T_10_App1Place={X 519.66385,Y 119.50261,Z 970.17229,A -180,B 0,C -180,S 2,T 2,E1 0,E2 0,E3 0,E4 0,E5 0,E6 0}
   E6POS P1_T_10_App2Place={X 519.66406,Y 119.50233,Z 820.17205,A 180,B 0,C 180,S 2,T 2,E1 0,E2 0,E3 0,E4 0,E5 0,E6 0}
   E6POS P1_T_10_Place={X 519.66406,Y 169.50233,Z 670.17205,A 180,B 0,C 180,S 2,T 2,E1 0,E2 0,E3 0,E4 0,E5 0,E6 0}
   E6POS P1_T_11_App1Place={X 519.66406,Y 169.50233,Z 970.17229,A 180,B 0,C 180,S 2,T 2,E1 0,E2 0,E3 0,E4 0,E5 0,E6 0}
   E6POS P1_T_11_App2Place={X 550.66406,Y 169.50233,Z 820.17205,A 180,B 0,C 180,S 2,T 2,E1 0,E2 0,E3 0,E4 0,E5 0,E6 0}
   E6POS P1_T_11_Place={X 550.66406,Y 169.50233,Z 670.17205,A 180,B 0,C 180,S 2,T 2,E1 0,E2 0,E3 0,E4 0,E5 0,E6 0}
   E6POS P1_T_12_App1Place={X 550.66406,Y 169.50233,Z 970.17229,A 180,B 0,C 180,S 2,T 2,E1 0,E2 0,E3 0,E4 0,E5 0,E6 0}
   E6POS P1_T_12_App2Place={X 581.66406,Y 169.50233,Z 820.17205,A 180,B 0,C 180,S 2,T 2,E1 0,E2 0,E3 0,E4 0,E5 0,E6 0}
   E6POS P1_T_12_Place={X 581.66406,Y 169.50233,Z 670.17205,A 180,B 0,C 180,S 2,T 2,E1 0,E2 0,E3 0,E4 0,E5 0,E6 0}

   ;ENDFOLD

   ;ENDFOLD
   ;FOLD Pallet2
   ;FOLD  MosaicoA_Pallet2

   E6POS P2_A_1_App1Place={X 392.37942,Y 496.91692,Z 990.1723,A -90,B 0,C 180,S 2,T 35,E1 0,E2 0,E3 0,E4 0,E5 0,E6 0}
   E6POS P2_A_1_App2Place={X 392.37943,Y 496.91703,Z 840.17238,A -90,B 0,C 180,S 2,T 35,E1 0,E2 0,E3 0,E4 0,E5 0,E6 0}
   E6POS P2_A_1_Place={X 303.26299,Y 448.70605,Z 670.17169,A -89.99997,B 0,C 180,S 2,T 35,E1 0,E2 0,E3 0,E4 0,E5 0,E6 0}
   E6POS P2_A_2_App1Place={X 717.00643,Y -14.89937,Z 990.1723,A -180,B 0,C 180,S 2,T 35,E1 0,E2 0,E3 0,E4 0,E5 0,E6 0}
   E6POS P2_A_2_App2Place={X 717.00728,Y -14.89935,Z 840.17238,A -180,B 0,C 180,S 2,T 35,E1 0,E2 0,E3 0,E4 0,E5 0,E6 0}
   E6POS P2_A_2_Place={X 567.90443,Y 149.73332,Z 670.17169,A -180,B 0,C -180,S 2,T 35,E1 0,E2 0,E3 0,E4 0,E5 0,E6 0}
   E6POS P2_A_3_App1Place={X 726.53443,Y 1132.46725,Z 990.1723,A -180,B 0,C 180,S 2,T 35,E1 0,E2 0,E3 0,E4 0,E5 0,E6 0}
   E6POS P2_A_3_App2Place={X 726.53453,Y 1132.4677,Z 840.17238,A -180,B 0,C 180,S 2,T 35,E1 0,E2 0,E3 0,E4 0,E5 0,E6 0}
   E6POS P2_A_3_Place={X 567.90337,Y 1005.46696,Z 670.17169,A -180,B 0,C 180,S 2,T 35,E1 0,E2 0,E3 0,E4 0,E5 0,E6 0}
   E6POS P2_A_4_App1Place={X 965.71856,Y 591.04703,Z 990.1723,A -90,B 0,C 180,S 2,T 35,E1 0,E2 0,E3 0,E4 0,E5 0,E6 0}
   E6POS P2_A_4_App2Place={X 965.71856,Y 591.04703,Z 840.17238,A -90,B 0,C 180,S 2,T 35,E1 0,E2 0,E3 0,E4 0,E5 0,E6 0}
   E6POS P2_A_4_Place={X 876.60642,Y 591.04703,Z 670.17169,A -90,B 0,C 180,S 2,T 35,E1 0,E2 0,E3 0,E4 0,E5 0,E6 0}
   E6POS P2_A_5_App1Place={X 964.37218,Y 240.84559,Z 990.1723,A -89.99997,B 0,C 180,S 2,T 35,E1 0,E2 0,E3 0,E4 0,E5 0,E6 0}
   E6POS P2_A_5_App2Place={X 964.37226,Y 240.84576,Z 840.17238,A -89.99997,B 0,C 180,S 2,T 35,E1 0,E2 0,E3 0,E4 0,E5 0,E6 0}
   E6POS P2_A_5_Place={X 875.26353,Y 446.44883,Z 670.17169,A -90,B 0,C -180,S 2,T 35,E1 0,E2 0,E3 0,E4 0,E5 0,E6 0}
   E6POS P2_A_6_App1Place={X 1159.8166,Y -10.11939,Z 990.1723,A -180,B 0,C -180,S 2,T 35,E1 0,E2 0,E3 0,E4 0,E5 0,E6 0}
   E6POS P2_A_6_App2Place={X 1159.81662,Y -10.11935,Z 840.17238,A -180,B 0,C 180,S 2,T 35,E1 0,E2 0,E3 0,E4 0,E5 0,E6 0}
   E6POS P2_A_6_Place={X 991.90433,Y 149.73252,Z 670.17169,A -180,B 0,C 180,S 2,T 35,E1 0,E2 0,E3 0,E4 0,E5 0,E6 0}
   E6POS P2_A_7_App1Place={X 847.78126,Y 1111.23569,Z 990.1723,A -180,B 0,C 180,S 2,T 35,E1 0,E2 0,E3 0,E4 0,E5 0,E6 0}
   E6POS P2_A_7_App2Place={X 847.78109,Y 1111.23506,Z 840.17238,A -180,B 0,C -180,S 2,T 35,E1 0,E2 0,E3 0,E4 0,E5 0,E6 0}
   E6POS P2_A_7_Place={X 991.90451,Y 1005.46652,Z 670.17169,A -180,B 0,C 180,S 2,T 35,E1 0,E2 0,E3 0,E4 0,E5 0,E6 0}
   E6POS P2_A_8_App1Place={X 54.19847,Y 589.83366,Z 990.1723,A -90,B 0,C 180,S 2,T 35,E1 0,E2 0,E3 0,E4 0,E5 0,E6 0}
   E6POS P2_A_8_App2Place={X 54.19848,Y 589.83349,Z 840.17238,A -90,B 0,C 180,S 2,T 35,E1 0,E2 0,E3 0,E4 0,E5 0,E6 0}
   E6POS P2_A_8_Place={X 168.87237,Y 591.04678,Z 670.17169,A -89.99997,B 0,C 180,S 2,T 35,E1 0,E2 0,E3 0,E4 0,E5 0,E6 0}

   ;ENDFOLD
   ;FOLD  MosaicoB_Pallet2

   E6POS P2_B_1_App1Place={X 696.23454,Y 929.21494,Z 986.29993,A -180,B 0,C 180,S 2,T 35,E1 0,E2 0,E3 0,E4 0,E5 0,E6 0}
   E6POS P2_B_1_App2Place={X 696.23427,Y 929.21551,Z 786.30015,A -180,B 0,C 180,S 2,T 35,E1 0,E2 0,E3 0,E4 0,E5 0,E6 0}
   E6POS P2_B_1_Place={X 567.29912,Y 1052.67757,Z 666.29996,A -180,B 0,C 180,S 2,T 35,E1 0,E2 0,E3 0,E4 0,E5 0,E6 0}
   E6POS P2_B_2_App1Place={X 562.37024,Y 346.47997,Z 986.29993,A -180,B 0,C 180,S 2,T 35,E1 0,E2 0,E3 0,E4 0,E5 0,E6 0}
   E6POS P2_B_2_App2Place={X 562.37047,Y 346.47964,Z 786.30015,A -180,B 0,C 180,S 2,T 35,E1 0,E2 0,E3 0,E4 0,E5 0,E6 0}
   E6POS P2_B_2_Place={X 433.43516,Y 269.94251,Z 666.29996,A -180,B 0,C -180,S 2,T 51,E1 0,E2 0,E3 0,E4 0,E5 0,E6 0}
   E6POS P2_B_3_App1Place={X 4.05094,Y 173.9296,Z 986.29993,A 90,B 0,C 180,S 2,T 35,E1 0,E2 0,E3 0,E4 0,E5 0,E6 0}
   E6POS P2_B_3_App2Place={X 4.05139,Y 177.15339,Z 786.30015,A 90,B 0,C 180,S 2,T 51,E1 0,E2 0,E3 0,E4 0,E5 0,E6 0}
   E6POS P2_B_3_Place={X 134.71509,Y 273.89023,Z 666.29996,A 90,B 0,C 180,S 2,T 51,E1 0,E2 0,E3 0,E4 0,E5 0,E6 0}
   E6POS P2_B_4_App1Place={X 1006.46579,Y 1126.41011,Z 986.29993,A -90,B 0,C 180,S 2,T 3,E1 0,E2 0,E3 0,E4 0,E5 0,E6 0}
   E6POS P2_B_4_App2Place={X 1006.46535,Y 1126.41022,Z 786.30015,A -90,B 0,C 180,S 2,T 3,E1 0,E2 0,E3 0,E4 0,E5 0,E6 0}
   E6POS P2_B_4_Place={X 866.11759,Y 921.41578,Z 666.29996,A -90,B 0,C -180,S 2,T 3,E1 0,E2 0,E3 0,E4 0,E5 0,E6 0}
   E6POS P2_B_5_App1Place={X 696.22115,Y 346.20661,Z 986.29993,A -180,B 0,C 180,S 2,T 35,E1 0,E2 0,E3 0,E4 0,E5 0,E6 0}
   E6POS P2_B_5_App2Place={X 696.22108,Y 346.20663,Z 786.30015,A -180,B 0,C 180,S 2,T 35,E1 0,E2 0,E3 0,E4 0,E5 0,E6 0}
   E6POS P2_B_5_Place={X 567.29973,Y 269.67394,Z 666.29996,A -180,B 0,C 180,S 2,T 35,E1 0,E2 0,E3 0,E4 0,E5 0,E6 0}
   E6POS P2_B_6_App1Place={X 562.37026,Y 929.4822,Z 986.29993,A -180,B 0,C 180,S 2,T 35,E1 0,E2 0,E3 0,E4 0,E5 0,E6 0}
   E6POS P2_B_6_App2Place={X 562.36973,Y 929.48268,Z 786.30015,A -180,B 0,C -180,S 2,T 35,E1 0,E2 0,E3 0,E4 0,E5 0,E6 0}
   E6POS P2_B_6_Place={X 433.43554,Y 1052.93855,Z 666.29996,A -180,B 0,C 180,S 2,T 35,E1 0,E2 0,E3 0,E4 0,E5 0,E6 0}
   E6POS P2_B_7_App1Place={X 30.66568,Y 1051.60367,Z 986.29993,A -90,B 0,C 180,S 2,T 35,E1 0,E2 0,E3 0,E4 0,E5 0,E6 0}
   E6POS P2_B_7_App2Place={X 30.66561,Y 1051.60341,Z 786.30015,A -90,B 0,C 180,S 2,T 35,E1 0,E2 0,E3 0,E4 0,E5 0,E6 0}
   E6POS P2_B_7_Place={X 175.26087,Y 921.40676,Z 666.29996,A -90,B 0,C 180,S 2,T 35,E1 0,E2 0,E3 0,E4 0,E5 0,E6 0}
   E6POS P2_B_8_App1Place={X 955.95613,Y 159.58069,Z 986.29993,A 90,B 0,C 180,S 2,T 35,E1 0,E2 0,E3 0,E4 0,E5 0,E6 0}
   E6POS P2_B_8_App2Place={X 955.95654,Y 159.58069,Z 786.30015,A 90,B 0,C 180,S 2,T 35,E1 0,E2 0,E3 0,E4 0,E5 0,E6 0}
   E6POS P2_B_8_Place={X 825.57189,Y 273.90166,Z 666.29996,A 90,B 0,C 180,S 2,T 35,E1 0,E2 0,E3 0,E4 0,E5 0,E6 0}

   ;ENDFOLD
   ;FOLD  MosaicoC1_Pallet2

   E6POS P2_C1_1_App1Place={X 585.89441,Y 217.9914,Z 986.28309,A -180,B 0,C 180,S 2,T 35,E1 0,E2 0,E3 0,E4 0,E5 0,E6 0}
   E6POS P2_C1_1_App2Place={X 585.89477,Y 217.99161,Z 836.28257,A -180,B 0,C -180,S 2,T 35,E1 0,E2 0,E3 0,E4 0,E5 0,E6 0}
   E6POS P2_C1_1_Place={X 512.66253,Y 90.04064,Z 666.30129,A -180,B 0,C 180,S 2,T 51,E1 0,E2 0,E3 0,E4 0,E5 0,E6 0}
   E6POS P2_C1_2_App1Place={X 585.89529,Y 456.99117,Z 986.28309,A -180,B 0,C 180,S 2,T 35,E1 0,E2 0,E3 0,E4 0,E5 0,E6 0}
   E6POS P2_C1_2_App2Place={X 585.89505,Y 456.99134,Z 836.28257,A -180,B 0,C -180,S 2,T 35,E1 0,E2 0,E3 0,E4 0,E5 0,E6 0}
   E6POS P2_C1_2_Place={X 512.66375,Y 329.04071,Z 666.30129,A -180,B 0,C 180,S 2,T 51,E1 0,E2 0,E3 0,E4 0,E5 0,E6 0}
   E6POS P2_C1_3_App1Place={X 606.92693,Y 689.18287,Z 986.28309,A -180,B 0,C 180,S 2,T 35,E1 0,E2 0,E3 0,E4 0,E5 0,E6 0}
   E6POS P2_C1_3_App2Place={X 606.92684,Y 689.18232,Z 836.28257,A -180,B 0,C 180,S 2,T 35,E1 0,E2 0,E3 0,E4 0,E5 0,E6 0}
   E6POS P2_C1_3_Place={X 537.74298,Y 568.04115,Z 666.30129,A -180,B 0,C 180,S 2,T 35,E1 0,E2 0,E3 0,E4 0,E5 0,E6 0}
   E6POS P2_C1_4_App1Place={X 606.92611,Y 1021.18252,Z 986.28309,A -180,B 0,C -180,S 2,T 35,E1 0,E2 0,E3 0,E4 0,E5 0,E6 0}
   E6POS P2_C1_4_App2Place={X 606.92631,Y 1021.18275,Z 836.28257,A -180,B 0,C 180,S 2,T 35,E1 0,E2 0,E3 0,E4 0,E5 0,E6 0}
   E6POS P2_C1_4_Place={X 537.74306,Y 900.04115,Z 666.30129,A -180,B 0,C -180,S 2,T 35,E1 0,E2 0,E3 0,E4 0,E5 0,E6 0}
   E6POS P2_C1_5_App1Place={X 606.20056,Y 212.00359,Z 986.28309,A -180,B 0,C 180,S 2,T 35,E1 0,E2 0,E3 0,E4 0,E5 0,E6 0}
   E6POS P2_C1_5_App2Place={X 606.20094,Y 212.00353,Z 836.28257,A -180,B 0,C 180,S 2,T 35,E1 0,E2 0,E3 0,E4 0,E5 0,E6 0}
   E6POS P2_C1_5_Place={X 539.21738,Y 90.04103,Z 666.30129,A -180,B 0,C -180,S 2,T 51,E1 0,E2 0,E3 0,E4 0,E5 0,E6 0}
   E6POS P2_C1_6_App1Place={X 606.20064,Y 544.00366,Z 986.28309,A -180,B 0,C 180,S 2,T 35,E1 0,E2 0,E3 0,E4 0,E5 0,E6 0}
   E6POS P2_C1_6_App2Place={X 606.20036,Y 544.00384,Z 836.28257,A -180,B 0,C 180,S 2,T 35,E1 0,E2 0,E3 0,E4 0,E5 0,E6 0}
   E6POS P2_C1_6_Place={X 539.2172,Y 422.04157,Z 666.30129,A -180,B 0,C 180,S 2,T 35,E1 0,E2 0,E3 0,E4 0,E5 0,E6 0}
   E6POS P2_C1_7_App1Place={X 516.90988,Y 854.03837,Z 986.28309,A -180,B 0,C 180,S 2,T 35,E1 0,E2 0,E3 0,E4 0,E5 0,E6 0}
   E6POS P2_C1_7_App2Place={X 516.9096,Y 854.03829,Z 836.28257,A -180,B 0,C 180,S 2,T 35,E1 0,E2 0,E3 0,E4 0,E5 0,E6 0}
   E6POS P2_C1_7_Place={X 516.90992,Y 754.0383,Z 666.30129,A -180,B 0,C -180,S 2,T 35,E1 0,E2 0,E3 0,E4 0,E5 0,E6 0}
   E6POS P2_C1_8_App1Place={X 516.90921,Y 1093.03906,Z 986.28309,A -180,B 0,C 180,S 2,T 35,E1 0,E2 0,E3 0,E4 0,E5 0,E6 0}
   E6POS P2_C1_8_App2Place={X 516.90967,Y 1093.03859,Z 836.28257,A -180,B 0,C 180,S 2,T 35,E1 0,E2 0,E3 0,E4 0,E5 0,E6 0}
   E6POS P2_C1_8_Place={X 516.90982,Y 993.03884,Z 666.30129,A -180,B 0,C -180,S 2,T 35,E1 0,E2 0,E3 0,E4 0,E5 0,E6 0}

   ;ENDFOLD
   ;FOLD  MosaicoE1_Pallet2

   E6POS P2_E1_1_App1Place={X 194.85179,Y 240.03154,Z 993.17112,A 90,B 0,C -180,S 2,T 35,E1 0,E2 0,E3 0,E4 0,E5 0,E6 0}
   E6POS P2_E1_1_App2Place={X 194.85179,Y 240.03149,Z 843.1711,A 90,B 0,C 180,S 2,T 35,E1 0,E2 0,E3 0,E4 0,E5 0,E6 0}
   E6POS P2_E1_1_Place={X 73.35816,Y 240.03167,Z 690.47496,A 90,B 0,C 180,S 2,T 51,E1 0,E2 0,E3 0,E4 0,E5 0,E6 0}
   E6POS P2_E1_2_App1Place={X 522.85182,Y 240.0316,Z 993.17112,A 90,B 0,C 180,S 2,T 35,E1 0,E2 0,E3 0,E4 0,E5 0,E6 0}
   E6POS P2_E1_2_App2Place={X 522.85174,Y 240.03121,Z 843.1711,A 90,B 0,C 180,S 2,T 35,E1 0,E2 0,E3 0,E4 0,E5 0,E6 0}
   E6POS P2_E1_2_Place={X 401.35813,Y 240.03144,Z 690.47496,A 90,B 0,C 180,S 2,T 51,E1 0,E2 0,E3 0,E4 0,E5 0,E6 0}
   E6POS P2_E1_3_App1Place={X 850.85189,Y 240.03178,Z 993.17112,A 90,B 0,C 180,S 2,T 35,E1 0,E2 0,E3 0,E4 0,E5 0,E6 0}
   E6POS P2_E1_3_App2Place={X 850.85169,Y 240.03128,Z 843.1711,A 90,B 0,C 180,S 2,T 35,E1 0,E2 0,E3 0,E4 0,E5 0,E6 0}
   E6POS P2_E1_3_Place={X 729.35887,Y 240.0316,Z 690.47496,A 90,B 0,C 180,S 2,T 51,E1 0,E2 0,E3 0,E4 0,E5 0,E6 0}
   E6POS P2_E1_4_App1Place={X 622.32104,Y 1010.79562,Z 993.17112,A 180,B 0,C 180,S 2,T 35,E1 0,E2 0,E3 0,E4 0,E5 0,E6 0}
   E6POS P2_E1_4_App2Place={X 622.32108,Y 1010.79584,Z 843.1711,A -180,B 0,C 180,S 2,T 35,E1 0,E2 0,E3 0,E4 0,E5 0,E6 0}
   E6POS P2_E1_4_Place={X 622.32108,Y 907.44031,Z 690.47496,A -180,B 0,C 180,S 2,T 35,E1 0,E2 0,E3 0,E4 0,E5 0,E6 0}
   E6POS P2_E1_5_App1Place={X 622.32111,Y 907.44046,Z 993.17112,A -180,B 0,C 180,S 2,T 35,E1 0,E2 0,E3 0,E4 0,E5 0,E6 0}
   E6POS P2_E1_5_App2Place={X 676.32064,Y 907.52752,Z 843.1711,A -180,B 0,C 180,S 2,T 35,E1 0,E2 0,E3 0,E4 0,E5 0,E6 0}
   E6POS P2_E1_5_Place={X 676.32052,Y 907.52694,Z 690.47496,A -180,B 0,C 180,S 2,T 35,E1 0,E2 0,E3 0,E4 0,E5 0,E6 0}
   E6POS P2_E1_6_App1Place={X 676.32064,Y 907.52752,Z 993.17112,A -180,B 0,C 180,S 2,T 35,E1 0,E2 0,E3 0,E4 0,E5 0,E6 0}
   E6POS P2_E1_6_App2Place={X 730.3205,Y 907.52691,Z 843.1711,A -180,B 0,C 180,S 2,T 35,E1 0,E2 0,E3 0,E4 0,E5 0,E6 0}
   E6POS P2_E1_6_Place={X 730.32055,Y 907.52712,Z 690.47496,A -180,B 0,C 180,S 2,T 35,E1 0,E2 0,E3 0,E4 0,E5 0,E6 0}
   E6POS P2_E1_7_App1Place={X 730.3205,Y 907.52691,Z 993.17112,A -180,B 0,C 180,S 2,T 35,E1 0,E2 0,E3 0,E4 0,E5 0,E6 0}
   E6POS P2_E1_7_App2Place={X 784.32058,Y 907.52713,Z 843.1711,A -180,B 0,C 180,S 2,T 35,E1 0,E2 0,E3 0,E4 0,E5 0,E6 0}
   E6POS P2_E1_7_Place={X 784.32065,Y 907.52737,Z 690.47496,A -180,B 0,C 180,S 2,T 35,E1 0,E2 0,E3 0,E4 0,E5 0,E6 0}
   E6POS P2_E1_8_App1Place={X 624.31125,Y 190.7954,Z 993.17112,A 180,B 0,C -180,S 2,T 35,E1 0,E2 0,E3 0,E4 0,E5 0,E6 0}
   E6POS P2_E1_8_App2Place={X 624.31125,Y 190.79541,Z 843.1711,A -180,B 0,C 180,S 2,T 35,E1 0,E2 0,E3 0,E4 0,E5 0,E6 0}

   E6POS P2_E1_8_Place={X 624.31203,Y 87.43905,Z 690.47496,A -180,B 0,C 180,S 2,T 35,E1 0,E2 0,E3 0,E4 0,E5 0,E6 0}
   E6POS P2_E1_9_App1Place={X 624.31193,Y 87.4387,Z 993.17112,A -180,B 0,C 180,S 2,T 35,E1 0,E2 0,E3 0,E4 0,E5 0,E6 0}
   E6POS P2_E1_9_App2Place={X 678.31177,Y 87.43866,Z 843.1711,A -180,B 0,C 180,S 2,T 35,E1 0,E2 0,E3 0,E4 0,E5 0,E6 0}

   E6POS P2_E1_9_Place={X 678.31185,Y 87.43891,Z 690.47496,A -180,B 0,C 180,S 2,T 35,E1 0,E2 0,E3 0,E4 0,E5 0,E6 0}
   E6POS P2_E1_10_App1Place={X 678.31177,Y 87.43866,Z 993.17112,A -180,B 0,C 180,S 2,T 35,E1 0,E2 0,E3 0,E4 0,E5 0,E6 0}
   E6POS P2_E1_10_App2Place={X 732.31118,Y 87.43893,Z 843.1711,A -180,B 0,C 180,S 2,T 35,E1 0,E2 0,E3 0,E4 0,E5 0,E6 0}

   E6POS P2_E1_10_Place={X 732.31137,Y 87.43945,Z 690.47496,A -180,B 0,C 180,S 2,T 35,E1 0,E2 0,E3 0,E4 0,E5 0,E6 0}
   E6POS P2_E1_11_App1Place={X 732.31118,Y 87.43893,Z 993.17112,A -180,B 0,C 180,S 2,T 35,E1 0,E2 0,E3 0,E4 0,E5 0,E6 0}
   E6POS P2_E1_11_App2Place={X 786.31144,Y 87.43887,Z 843.1711,A -180,B 0,C 180,S 2,T 35,E1 0,E2 0,E3 0,E4 0,E5 0,E6 0}

   E6POS P2_E1_11_Place={X 786.31151,Y 87.43905,Z 690.47496,A -180,B 0,C 180,S 2,T 35,E1 0,E2 0,E3 0,E4 0,E5 0,E6 0}
   E6POS P2_E1_12_App1Place={X 838.55893,Y 1064.39321,Z 993.17112,A -90,B 0,C -180,S 2,T 3,E1 0,E2 0,E3 0,E4 0,E5 0,E6 0}
   E6POS P2_E1_12_App2Place={X 838.55901,Y 1064.39353,Z 843.1711,A -90,B 0,C 180,S 2,T 3,E1 0,E2 0,E3 0,E4 0,E5 0,E6 0}

   E6POS P2_E1_12_Place={X 938.55894,Y 964.39354,Z 690.47496,A -90,B 0,C 180,S 2,T 3,E1 0,E2 0,E3 0,E4 0,E5 0,E6 0}
   E6POS P2_E1_13_App1Place={X 510.55806,Y 1064.39378,Z 993.17112,A -89.99997,B 0,C -180,S 2,T 3,E1 0,E2 0,E3 0,E4 0,E5 0,E6 0}
   E6POS P2_E1_13_App2Place={X 510.55802,Y 1064.39347,Z 843.1711,A -89.99997,B 0,C 180,S 2,T 3,E1 0,E2 0,E3 0,E4 0,E5 0,E6 0}

   E6POS P2_E1_13_Place={X 610.5583,Y 964.39342,Z 690.47496,A -89.99997,B 0,C 180,S 2,T 3,E1 0,E2 0,E3 0,E4 0,E5 0,E6 0}
   E6POS P2_E1_14_App1Place={X 182.55871,Y 1064.39361,Z 993.17112,A -90,B 0,C -180,S 2,T 35,E1 0,E2 0,E3 0,E4 0,E5 0,E6 0}
   E6POS P2_E1_14_App2Place={X 182.55871,Y 1064.39336,Z 843.1711,A -90,B 0,C 180,S 2,T 35,E1 0,E2 0,E3 0,E4 0,E5 0,E6 0}

   E6POS P2_E1_14_Place={X 282.55806,Y 964.39307,Z 690.47496,A -89.99997,B 0,C 180,S 2,T 3,E1 0,E2 0,E3 0,E4 0,E5 0,E6 0}

   ;ENDFOLD
   ;FOLD  MosaicoE2_Pallet2

   E6POS P2_E2_1_App1Place={X 194.85179,Y 240.03154,Z 953.17112,A 90,B 0,C -180,S 2,T 35,E1 0,E2 0,E3 0,E4 0,E5 0,E6 0}
   E6POS P2_E2_1_App2Place={X 194.85179,Y 240.03149,Z 803.1711,A 90,B 0,C 180,S 2,T 51,E1 0,E2 0,E3 0,E4 0,E5 0,E6 0}
   E6POS P2_E2_1_Place={X 73.35816,Y 240.03167,Z 650.47496,A 90,B 0,C 180,S 2,T 51,E1 0,E2 0,E3 0,E4 0,E5 0,E6 0}
   E6POS P2_E2_2_App1Place={X 522.85182,Y 240.0316,Z 953.17112,A 90,B 0,C 180,S 2,T 35,E1 0,E2 0,E3 0,E4 0,E5 0,E6 0}
   E6POS P2_E2_2_App2Place={X 522.85174,Y 240.03121,Z 803.1711,A 90,B 0,C 180,S 2,T 35,E1 0,E2 0,E3 0,E4 0,E5 0,E6 0}
   E6POS P2_E2_2_Place={X 401.35813,Y 240.03144,Z 650.47496,A 90,B 0,C 180,S 2,T 51,E1 0,E2 0,E3 0,E4 0,E5 0,E6 0}
   E6POS P2_E2_3_App1Place={X 850.85189,Y 240.03178,Z 953.17112,A 90,B 0,C 180,S 2,T 35,E1 0,E2 0,E3 0,E4 0,E5 0,E6 0}
   E6POS P2_E2_3_App2Place={X 850.85169,Y 240.03128,Z 803.1711,A 90,B 0,C 180,S 2,T 35,E1 0,E2 0,E3 0,E4 0,E5 0,E6 0}
   E6POS P2_E2_3_Place={X 729.35887,Y 240.0316,Z 650.47496,A 90,B 0,C 180,S 2,T 51,E1 0,E2 0,E3 0,E4 0,E5 0,E6 0}
   E6POS P2_E2_4_App1Place={X 622.32104,Y 1010.79562,Z 953.17112,A 180,B 0,C -180,S 2,T 35,E1 0,E2 0,E3 0,E4 0,E5 0,E6 0}
   E6POS P2_E2_4_App2Place={X 622.32108,Y 1010.79584,Z 803.1711,A -180,B 0,C 180,S 2,T 35,E1 0,E2 0,E3 0,E4 0,E5 0,E6 0}
   E6POS P2_E2_4_Place={X 622.32108,Y 907.44031,Z 650.47496,A -180,B 0,C 180,S 2,T 35,E1 0,E2 0,E3 0,E4 0,E5 0,E6 0}
   E6POS P2_E2_5_App1Place={X 622.32111,Y 907.44046,Z 953.17112,A -180,B 0,C 180,S 2,T 35,E1 0,E2 0,E3 0,E4 0,E5 0,E6 0}
   E6POS P2_E2_5_App2Place={X 676.32064,Y 907.52752,Z 803.1711,A -180,B 0,C 180,S 2,T 35,E1 0,E2 0,E3 0,E4 0,E5 0,E6 0}
   E6POS P2_E2_5_Place={X 676.32052,Y 907.52694,Z 650.47496,A -180,B 0,C 180,S 2,T 35,E1 0,E2 0,E3 0,E4 0,E5 0,E6 0}
   E6POS P2_E2_6_App1Place={X 676.32064,Y 907.52752,Z 953.17112,A -180,B 0,C 180,S 2,T 35,E1 0,E2 0,E3 0,E4 0,E5 0,E6 0}
   E6POS P2_E2_6_App2Place={X 730.3205,Y 907.52691,Z 803.1711,A -180,B 0,C 180,S 2,T 35,E1 0,E2 0,E3 0,E4 0,E5 0,E6 0}
   E6POS P2_E2_6_Place={X 730.32055,Y 907.52712,Z 650.47496,A -180,B 0,C 180,S 2,T 35,E1 0,E2 0,E3 0,E4 0,E5 0,E6 0}
   E6POS P2_E2_7_App1Place={X 730.3205,Y 907.52691,Z 953.17112,A -180,B 0,C 180,S 2,T 35,E1 0,E2 0,E3 0,E4 0,E5 0,E6 0}
   E6POS P2_E2_7_App2Place={X 784.32058,Y 907.52713,Z 803.1711,A -180,B 0,C 180,S 2,T 35,E1 0,E2 0,E3 0,E4 0,E5 0,E6 0}
   E6POS P2_E2_7_Place={X 784.32065,Y 907.52737,Z 650.47496,A -180,B 0,C 180,S 2,T 35,E1 0,E2 0,E3 0,E4 0,E5 0,E6 0}
   E6POS P2_E2_8_App1Place={X 624.31125,Y 190.7954,Z 953.17112,A 180,B 0,C -180,S 2,T 35,E1 0,E2 0,E3 0,E4 0,E5 0,E6 0}
   E6POS P2_E2_8_App2Place={X 624.31125,Y 190.79541,Z 803.1711,A -180,B 0,C 180,S 2,T 35,E1 0,E2 0,E3 0,E4 0,E5 0,E6 0}
   E6POS P2_E2_8_Place={X 624.31203,Y 87.43905,Z 650.47496,A -180,B 0,C 180,S 2,T 51,E1 0,E2 0,E3 0,E4 0,E5 0,E6 0}
   E6POS P2_E2_9_App1Place={X 624.31193,Y 87.4387,Z 953.17112,A -180,B 0,C 180,S 2,T 35,E1 0,E2 0,E3 0,E4 0,E5 0,E6 0}
   E6POS P2_E2_9_App2Place={X 678.31177,Y 87.43866,Z 803.1711,A -180,B 0,C 180,S 2,T 35,E1 0,E2 0,E3 0,E4 0,E5 0,E6 0}
   E6POS P2_E2_9_Place={X 678.31185,Y 87.43891,Z 650.47496,A -180,B 0,C -180,S 2,T 51,E1 0,E2 0,E3 0,E4 0,E5 0,E6 0}
   E6POS P2_E2_10_App1Place={X 678.31177,Y 87.43866,Z 953.17112,A -180,B 0,C 180,S 2,T 35,E1 0,E2 0,E3 0,E4 0,E5 0,E6 0}
   E6POS P2_E2_10_App2Place={X 732.31118,Y 87.43893,Z 803.1711,A -180,B 0,C 180,S 2,T 35,E1 0,E2 0,E3 0,E4 0,E5 0,E6 0}
   E6POS P2_E2_10_Place={X 732.31137,Y 87.43945,Z 650.47496,A -180,B 0,C 180,S 2,T 35,E1 0,E2 0,E3 0,E4 0,E5 0,E6 0}
   E6POS P2_E2_11_App1Place={X 732.31118,Y 87.43893,Z 953.17112,A -180,B 0,C 180,S 2,T 35,E1 0,E2 0,E3 0,E4 0,E5 0,E6 0}
   E6POS P2_E2_11_App2Place={X 786.31144,Y 87.43887,Z 803.1711,A -180,B 0,C -180,S 2,T 35,E1 0,E2 0,E3 0,E4 0,E5 0,E6 0}
   E6POS P2_E2_11_Place={X 786.31151,Y 87.43905,Z 650.47496,A -180,B 0,C -180,S 2,T 35,E1 0,E2 0,E3 0,E4 0,E5 0,E6 0}
   E6POS P2_E2_12_App1Place={X 838.55893,Y 1064.39321,Z 953.17112,A -90,B 0,C -180,S 2,T 3,E1 0,E2 0,E3 0,E4 0,E5 0,E6 0}
   E6POS P2_E2_12_App2Place={X 838.55901,Y 1064.39353,Z 803.1711,A -90,B 0,C 180,S 2,T 3,E1 0,E2 0,E3 0,E4 0,E5 0,E6 0}

   E6POS P2_E2_12_Place={X 938.55894,Y 964.39354,Z 650.47496,A -90,B 0,C 180,S 2,T 3,E1 0,E2 0,E3 0,E4 0,E5 0,E6 0}
   E6POS P2_E2_13_App1Place={X 510.55806,Y 1064.39378,Z 953.17112,A -89.99997,B 0,C -180,S 2,T 3,E1 0,E2 0,E3 0,E4 0,E5 0,E6 0}
   E6POS P2_E2_13_App2Place={X 510.55802,Y 1064.39347,Z 803.1711,A -89.99997,B 0,C 180,S 2,T 3,E1 0,E2 0,E3 0,E4 0,E5 0,E6 0}

   E6POS P2_E2_13_Place={X 610.5583,Y 964.39342,Z 650.47496,A -89.99997,B 0,C 180,S 2,T 3,E1 0,E2 0,E3 0,E4 0,E5 0,E6 0}
   E6POS P2_E2_14_App1Place={X 182.55871,Y 1064.39361,Z 953.17112,A -90,B 0,C -180,S 2,T 35,E1 0,E2 0,E3 0,E4 0,E5 0,E6 0}
   E6POS P2_E2_14_App2Place={X 182.55871,Y 1064.39336,Z 803.1711,A -90,B 0,C 180,S 2,T 35,E1 0,E2 0,E3 0,E4 0,E5 0,E6 0}

   E6POS P2_E2_14_Place={X 282.55806,Y 964.39307,Z 650.47496,A -89.99997,B 0,C 180,S 2,T 3,E1 0,E2 0,E3 0,E4 0,E5 0,E6 0}

   ;ENDFOLD
   ;FOLD  MosaicoF_Pallet2

   E6POS P2_F_1_App1Place={X 185.71038,Y 503.84687,Z 990.17128,A -89.99997,B 0,C -180,S 2,T 35,E1 0,E2 0,E3 0,E4 0,E5 0,E6 0}
   E6POS P2_F_1_App2Place={X 185.71037,Y 503.84729,Z 840.17131,A -89.99997,B 0,C 180,S 2,T 35,E1 0,E2 0,E3 0,E4 0,E5 0,E6 0}
   E6POS P2_F_1_Place={X 59.05642,Y 604.23198,Z 654.93708,A -89.99997,B 0,C 180,S 2,T 35,E1 0,E2 0,E3 0,E4 0,E5 0,E6 0}
   E6POS P2_F_2_App1Place={X 484.71026,Y 503.84719,Z 990.17128,A -89.99997,B 0,C -180,S 2,T 3,E1 0,E2 0,E3 0,E4 0,E5 0,E6 0}
   E6POS P2_F_2_App2Place={X 484.71027,Y 503.84725,Z 840.17131,A -89.99997,B 0,C 180,S 2,T 3,E1 0,E2 0,E3 0,E4 0,E5 0,E6 0}
   E6POS P2_F_2_Place={X 358.05527,Y 604.23504,Z 654.93708,A -89.99997,B 0,C 180,S 2,T 3,E1 0,E2 0,E3 0,E4 0,E5 0,E6 0}
   E6POS P2_F_3_App1Place={X 783.33989,Y 500.30983,Z 990.17128,A -90,B 0,C -180,S 2,T 3,E1 0,E2 0,E3 0,E4 0,E5 0,E6 0}
   E6POS P2_F_3_App2Place={X 783.33995,Y 500.31005,Z 840.17131,A -90,B 0,C 180,S 2,T 3,E1 0,E2 0,E3 0,E4 0,E5 0,E6 0}
   E6POS P2_F_3_Place={X 657.05567,Y 600.73453,Z 654.93708,A -90,B 0,C 180,S 2,T 3,E1 0,E2 0,E3 0,E4 0,E5 0,E6 0}
   E6POS P2_F_4_App1Place={X 981.33997,Y 500.31013,Z 990.17128,A -90,B 0,C -180,S 2,T 3,E1 0,E2 0,E3 0,E4 0,E5 0,E6 0}
   E6POS P2_F_4_App2Place={X 981.33982,Y 500.30975,Z 840.17131,A -90,B 0,C 180,S 2,T 3,E1 0,E2 0,E3 0,E4 0,E5 0,E6 0}
   E6POS P2_F_4_Place={X 855.0547,Y 600.73492,Z 654.93708,A -90,B 0,C 180,S 2,T 3,E1 0,E2 0,E3 0,E4 0,E5 0,E6 0}
   E6POS P2_F_5_App1Place={X 185.33937,Y 495.81022,Z 990.17128,A -90,B 0,C 180,S 2,T 35,E1 0,E2 0,E3 0,E4 0,E5 0,E6 0}
   E6POS P2_F_5_App2Place={X 185.33937,Y 495.81034,Z 840.17131,A -90,B 0,C 180,S 2,T 35,E1 0,E2 0,E3 0,E4 0,E5 0,E6 0}
   E6POS P2_F_5_Place={X 59.05866,Y 596.22286,Z 654.93708,A -90,B 0,C 180,S 2,T 35,E1 0,E2 0,E3 0,E4 0,E5 0,E6 0}
   E6POS P2_F_6_App1Place={X 383.33975,Y 495.81046,Z 990.17128,A -90,B 0,C -180,S 2,T 3,E1 0,E2 0,E3 0,E4 0,E5 0,E6 0}
   E6POS P2_F_6_App2Place={X 383.33973,Y 495.81031,Z 840.17131,A -90,B 0,C 180,S 2,T 3,E1 0,E2 0,E3 0,E4 0,E5 0,E6 0}
   E6POS P2_F_6_Place={X 257.05855,Y 596.22277,Z 654.93708,A -90,B 0,C 180,S 2,T 3,E1 0,E2 0,E3 0,E4 0,E5 0,E6 0}
   E6POS P2_F_7_App1Place={X 581.71087,Y 500.34668,Z 990.17128,A -90,B 0,C -180,S 2,T 3,E1 0,E2 0,E3 0,E4 0,E5 0,E6 0}
   E6POS P2_F_7_App2Place={X 581.71089,Y 500.3468,Z 840.17131,A -90,B 0,C 180,S 2,T 3,E1 0,E2 0,E3 0,E4 0,E5 0,E6 0}
   E6POS P2_F_7_Place={X 455.05485,Y 600.73514,Z 654.93708,A -90,B 0,C 180,S 2,T 3,E1 0,E2 0,E3 0,E4 0,E5 0,E6 0}
   E6POS P2_F_8_App1Place={X 880.71048,Y 500.34632,Z 990.17128,A -90,B 0,C 180,S 2,T 3,E1 0,E2 0,E3 0,E4 0,E5 0,E6 0}
   E6POS P2_F_8_App2Place={X 880.7105,Y 500.34636,Z 840.17131,A -90,B 0,C 180,S 2,T 3,E1 0,E2 0,E3 0,E4 0,E5 0,E6 0}
   E6POS P2_F_8_Place={X 754.05499,Y 600.73496,Z 654.93708,A -90,B 0,C 180,S 2,T 3,E1 0,E2 0,E3 0,E4 0,E5 0,E6 0}

   ;ENDFOLD
   ;FOLD  MosaicoG_Pallet2

